(* Logix 5000 project; controller cal1632 1756-L62 rev 16.20; software revision 16.05; part 2 of 57 *)

ADD_ON_INSTRUCTION SYS_RPM_TO_SPEED   (* revision 1.0 *)
VAR_INPUT
   IN_gear_ratio : REAL; {required}
   IN_roll_diameter : REAL; {required}
   IN_vfd_fb_rpm : REAL; {required}
END_VAR
VAR_OUTPUT
   OUT_surface_speed_fb : REAL; {required}
END_VAR
VAR
   no_diameter : BOOL;
END_VAR

ROUTINE Logic   (* ladder *)
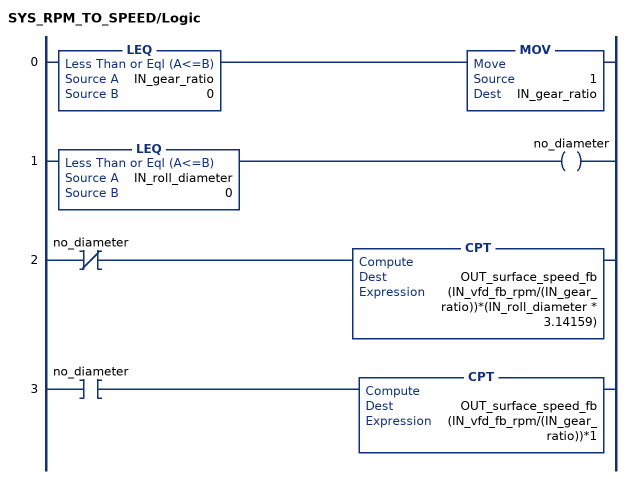
   0: LEQ(IN_gear_ratio,0)MOV(1,IN_gear_ratio);
   1: LEQ(IN_roll_diameter,0)OTE(no_diameter);
   2: XIO(no_diameter)CPT(OUT_surface_speed_fb,(IN_vfd_fb_rpm/(IN_gear_ratio))*(IN_roll_diameter * 3.14159));
   3: XIC(no_diameter)CPT(OUT_surface_speed_fb,(IN_vfd_fb_rpm/(IN_gear_ratio))*1);
END_ROUTINE
END_ADD_ON_INSTRUCTION

ADD_ON_INSTRUCTION SYS_SCP   (* revision 1.0 *)
VAR_INPUT
   Input : REAL; {required}
   Input_Min : REAL; {required}
   Input_Max : REAL; {required}
   Output_Min : REAL; {required}
   Output_Max : REAL; {required}
END_VAR
VAR_OUTPUT
   Output : REAL; {required}
   Fault : BOOL;
END_VAR
VAR
   m : REAL;
   b : REAL;
   X1 : REAL;
   X2 : REAL;
   Y1 : REAL;
   Y2 : REAL;
   X3 : REAL;
   Y3 : REAL;
END_VAR

ROUTINE Logic   (* ladder *)
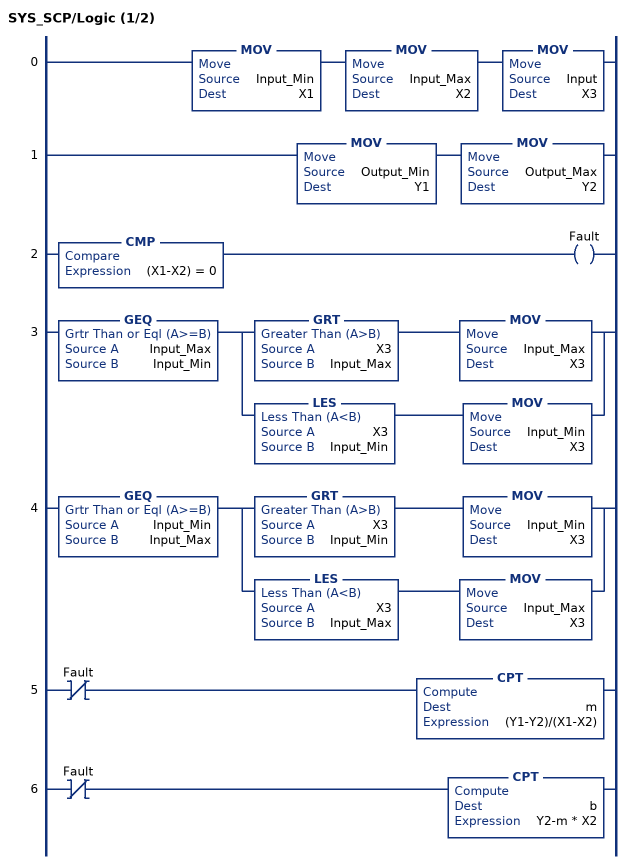
   0: MOV(Input_Min,X1)MOV(Input_Max,X2)MOV(Input,X3);
   1: MOV(Output_Min,Y1)MOV(Output_Max,Y2);
   2: CMP((X1-X2) = 0)OTE(Fault);
   3: GEQ(Input_Max,Input_Min)[GRT(X3,Input_Max) MOV(Input_Max,X3) ,LES(X3,Input_Min) MOV(Input_Min,X3) ];
   4: GEQ(Input_Min,Input_Max)[GRT(X3,Input_Min) MOV(Input_Min,X3) ,LES(X3,Input_Max) MOV(Input_Max,X3) ];
   5: XIO(Fault)CPT(m,(Y1-Y2)/(X1-X2));
   6: XIO(Fault)CPT(b,Y2-m * X2);
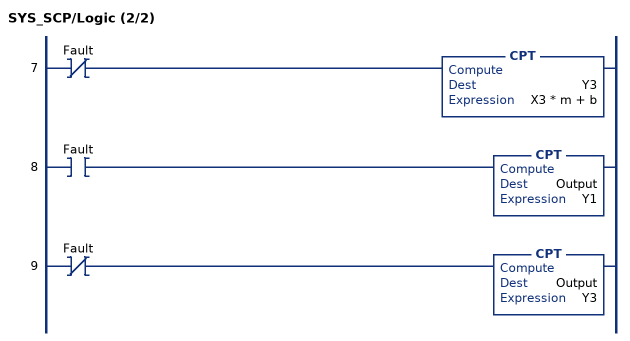
   7: XIO(Fault)CPT(Y3,X3 * m + b);
   8: XIC(Fault)CPT(Output,Y1);
   9: XIO(Fault)CPT(Output,Y3);
END_ROUTINE
END_ADD_ON_INSTRUCTION

ADD_ON_INSTRUCTION SYS_SPEED_TO_VFD   (* revision 1.0 *)
VAR_INPUT
   IN_gear_ratio : REAL; {required}
   IN_roll_diameter : REAL; {required}
   IN_selected_speed : REAL; {required}
END_VAR
VAR_OUTPUT
   OUT_surface_speed_rpm : REAL; {required}
END_VAR

ROUTINE Logic   (* ladder *)
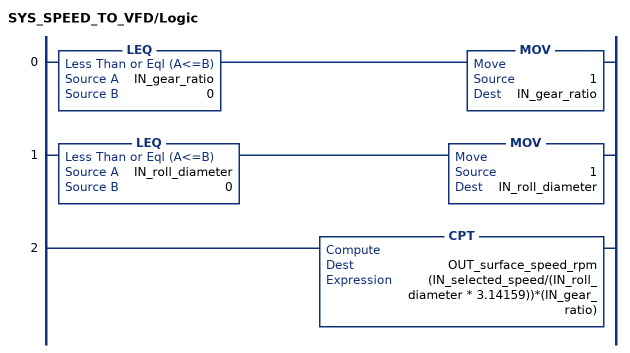
   0: LEQ(IN_gear_ratio,0)MOV(1,IN_gear_ratio);
   1: LEQ(IN_roll_diameter,0)MOV(1,IN_roll_diameter);
   2: CPT(OUT_surface_speed_rpm,(IN_selected_speed/(IN_roll_diameter * 3.14159))*(IN_gear_ratio));
END_ROUTINE
END_ADD_ON_INSTRUCTION

ADD_ON_INSTRUCTION SYS_Toggle   (* revision 1.0 *)
VAR_INPUT
   in_pb : BOOL; {required}
END_VAR
VAR_IN_OUT
   out_state : BOOL; {required}
END_VAR
VAR_INPUT
   toggle_state : BOOL; {visible}
END_VAR
VAR
   ons : DINT;
   toggle_select_deselct : BOOL;
END_VAR

ROUTINE Logic   (* ladder *)
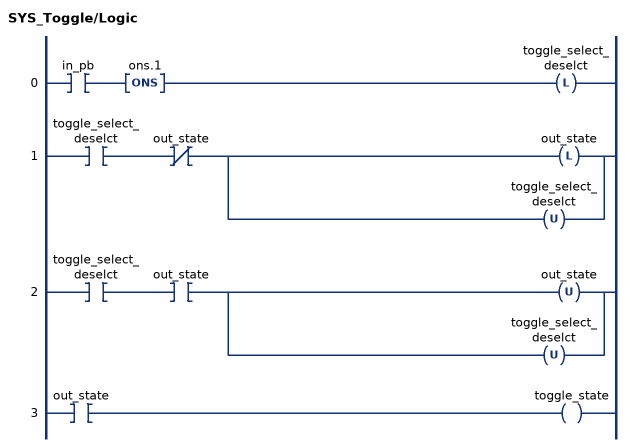
   0: XIC(in_pb)ONS(ons.1)OTL(toggle_select_deselct);
   1: XIC(toggle_select_deselct)XIO(out_state)[OTL(out_state) ,OTU(toggle_select_deselct) ];
   2: XIC(toggle_select_deselct)XIC(out_state)[OTU(out_state) ,OTU(toggle_select_deselct) ];
   3: XIC(out_state)OTE(toggle_state);
END_ROUTINE
END_ADD_ON_INSTRUCTION

VAR_GLOBAL   (* controller tags *)
   aaa_prs : REAL := 60.0;
   AFI : BOOL;
   FAULT : BOOL;
   HMI : BOOL;
   metering_roll : TIMER := (PRE := 4500);
   metering_roll_alarm : TIMER := (PRE := 4500);
   metering_roll_close : TIMER := (PRE := 5000);
   P00_VFD_Sprng_PID : PID := (SP := 25.0, OUT := 10.0);
   p01_ai_lc_4 : REAL := 0.95815146;
   p01_ai_prs : REAL := -2.5;
   p01_ai_tc : REAL := 132.4;
   p01_di_edge_ctrl_estop_active : BOOL;
   p01_di_estop_1_tripped : BOOL := 1;
   p01_di_estop_2_tripped : BOOL := 1;
   p01_di_estop_reset : BOOL;
   p01_di_impreg_estop_active : BOOL;
   p01_di_letoff_estop_active : BOOL;
   p01_di_lof_acc_estop_active : BOOL;
   p01_di_main_hmi_estop : BOOL;
   p01_di_rope_sw_1_active : BOOL;
   p01_di_rope_sw_2_active : BOOL;
   p01_di_rope_sw_3_active : BOOL;
   p01_di_rope_sw_4_active : BOOL;
   p01_di_rope_sw_5_active : BOOL;
   p01_di_rope_sw_6_active : BOOL;
   p01_di_rope_sw_7_active : BOOL;
   p01_di_rope_sw_8_active : BOOL;
   p01_di_splice_estop_active : BOOL;
   p01_di_ts2_estop_active : BOOL;
   p01_di_winder_estop_active : BOOL;
   p01_dint_to_hmi : DINT[16] := ([0] := 643, [1] := 2, [3] := 128, [4] := 2, [6] := 133, [7] := 2, [8] := 5, [9] := 9, [14] := 18806);
   p01_int_from_oxidizer : INT[10] := ([0] := 528, [1] := 2, [2] := 93, [3] := 121, [4] := 1688, [5] := 1689, [6] := 214, [7] := 88, [8] := 1385, [9] := 1608); {produced}
   p01_int_to_oxidizer : INT;
   p01_param_fan_zero_speed : REAL := 0.1;
   p01_param_heater_hl : REAL := 785.0;
   p01_param_master_accel : REAL := 0.5;
   p01_param_master_decel : REAL := 2.5;
   p01_param_master_jog_accel : REAL := 10.0;
   p01_param_master_jog_decel : REAL := 20.0;
   p01_param_master_jog_speed : REAL := 13.0;
   p01_param_min_start_tension : REAL := 10.0;
   p01_param_mtr_over_speed_pct : REAL := 0.4;
   p01_param_open_oven_exh_sp : REAL := 300.0;
   p01_param_open_oven_recirc_sp : REAL := 300.0;
   p01_param_open_oven_temp : REAL := 80.0;
   p01_param_oven_timer_presets : DINT[32] := ([1] := 500, [2] := 10000, [3] := 20000, [6] := 5000, [8] := 1000, [9] := 1000, [10] := 1000, [11] := 5000, [14] := 10000, [16] := 1000, [17] := 90000, [18] := 1500, [19] := 1000, [21] := 1000, [22] := 1000, [23] := 2000, [24] := 5000, [25] := 5000, [26] := 15000, [27] := 500, [28] := 30000, [31] := 500);
   p01_param_process_air_hl : REAL := 500.0;
   p01_param_process_air_max : REAL := 480.0;
   p01_param_slow_speed_sp : REAL := 2.0;
   p01_param_start_delay : REAL := 6.5;
   p01_param_temp_limit : REAL := 120.0;
   p01_param_tension_deviation : REAL := 5.0;
   p01_param_turret_dia_ft : REAL := 3.2;
   p01_r15_footage_ft : REAL;
   p01_real_to_hmi : REAL[112] := ([1] := 13.0, [11] := 92.0, [12] := 128.0, [13] := 1690.0, [14] := 1694.0, [15] := 220.0, [16] := 88.0, [17] := 1370.0, [18] := 1621.0, [19] := 8953.26);
   p01_recipe_active : recipe := (name := 'CP:F-555-S:1KPW:JOBY.csv', master_line_speed := 10.0, zone_1.recirc_sp := 1000.0, zone_1.exhaust_sp := 900.0, zone_1.temp_sp := 225.0, zone_2.recirc_sp := 1000.0, zone_2.exhaust_sp := 900.0, zone_2.temp_sp := 225.0, zone_3.recirc_sp := 1000.0, zone_3.exhaust_sp := 900.0, zone_3.temp_sp := 70.0, line_speed_sp := 13.0, letoff_tension_sp := 15.0, acc_tension_sp := 60.0, acc_fill_pressure_sp := 10.0, acc_counter_pressure_sp := 10.0, cure_time_sp := 55.0, platen_temp_sp := 450.0, impreg_gap_sp := 0.0175, impreg_supply_speed_sp := 1200.0, ts1_tension_sp := 60.0, adv_cooling_temp_sp := 65.0, ts2_tension_sp := 60.0, lower_poly_tension_sp := 3.0, lower_poly_b_tension_sp := 3.0, upper_poly_tension_sp := 3.0, upper_poly_b_tension_sp := 3.0, winder_tension_sp := 70.0, winder_torque_sp := 100.0, tension_deviation_sp := 15.0);
   p01_sys_enc : SYS_ENC := (IN_State := 3, OUT_Status := 1);
   p01_sys_lc : Limit_Clamp := (max := 100.0);
   p01_sys_scp : SYS_SCP := (Input := 12760.0, Input_Max := 30840.0, Output_Max := 50.0, Output := 20.68742);
   p01r01 : routine := (comment := 7);
   p01r02 : routine := (comment := -1073741569, fault := 32768, fault_ack := 32768);
   p01r02_all_fans_stopped : BOOL := 1;
   p01r02_batch_run_time : DINT := 24;
   p01r02_batch_run_time_hrs : DINT := 18806;
   p01r02_do_buzzer : BOOL;
   p01r02_do_buzzer_LINE : BOOL := 1;
   p01r02_do_green_stack_light_lel : BOOL := 1;
   p01r02_do_green_stack_light_LINE : BOOL;
   p01r02_do_horn : BOOL;
   p01r02_do_red_stack_light : BOOL;
   p01r02_do_red_stack_light_LINE : BOOL := 1;
   p01r02_do_yellow_stack_light : BOOL;
   p01r02_do_yellow_stack_light_LINE : BOOL := 1;
   p01r02_ethernet_comm : DINT := 491519;
   p01r02_fault_exists : BOOL;
   p01r02_flash_bit : BOOL;
   p01r02_flash_timer_off : TIMER := (PRE := 1000);
   p01r02_flash_timer_on : TIMER := (PRE := 1000, ACC := 979, EN := 1, TT := 1);
   p01r02_horn : BOOL := 1;
   p01r02_plc_faults : DINT := 16;
   p01r02_plc_scan_time : DINT := 30386;
   p01r02_plc_scan_time_in_sec : REAL := 0.030494;
   p01r02_timer_batch : TIMER := (PRE := 60000);
   p01r02_timer_fault : TIMER[25] := ([15].ACC := 31, [15].EN := 1, [15].DN := 1);
   p01r02_timer_half_second_off : TIMER := (PRE := 300);
   p01r02_timer_half_second_on : TIMER := (PRE := 300, ACC := 305, EN := 1, DN := 1);
   p01r02_timer_second : TIMER[2] := ([0].PRE := 1000, [0].ACC := 1009, [0].EN := 1, [0].DN := 1, [1].PRE := 1000, [1].ACC := 551, [1].EN := 1, [1].TT := 1);
   p01r02_timer_warning : TIMER[4];
   p01r02_unack_fault : BOOL;
   p01r02_unack_warning : BOOL := 1;
   p01r02_vfd_comm_2 : DINT[50] := ([0] := 16897, [1] := 16897, [2] := 16897, [3] := 16897, [4] := 16897, [5] := 16897, [6] := 16897, [7] := 16897, [8] := 16897, [9] := 16897, [10] := 16897, [11] := 16897, [12] := 16897, [13] := 16897, [14] := 16897, [15] := 4096, [16] := 16897, [17] := 16897, [18] := 16897);
   p01r02_warnings_exists : BOOL := 1;
   p01r03 : routine := (comment := -1073741793);
   p01r03_lc3_ave_ctrl : CONTROL := (LEN := 19);
   p01r03_oxidizer_prs : SYS_SCP := (Input_Max := 30840.0, Output_Min := -2.5, Output_Max := 2.5, Output := -2.5);
   p01r03_prs_input_max : REAL := 30840.0;
   p01r03_prs_input_min : REAL;
   p01r03_prs_output_max : REAL := 2.5;
   p01r03_prs_output_min : REAL := -2.5;
   p01r03_timer_fault : TIMER[4];
   p01r03_timer_warning : TIMER[4];
   p01r04 : routine := (comment := -1073741793);
   p01r04_LFL_warning : BOOL;
   p01r04_Temp_deviation_warning : BOOL := 1;
   p01r04_timer_fault : TIMER[4];
   p01r04_timer_warning : TIMER[4];
   p01r05 : routine := (comment := -1073741761);
   p01r05_enc : SYS_ENC;
   p01r05_timer_fault : TIMER[4];
   p01r05_timer_warning : TIMER[4];
   p01r06 : routine := (comment := -1073741572);
   p01r06_timer_fault : TIMER[4];
   p01r06_timer_warning : TIMER[4];
   p01r07 : routine := (comment := -1073741761);
   p01r07_timer_fault : TIMER[4];
   p01r07_timer_warning : TIMER[4];
   p01r08 : routine := (comment := -1073741761);
   p01r08_timer_fault : TIMER[4];
   p01r08_timer_warning : TIMER[4];
   p01r09 : routine := (comment := -1073741009, oneshot := 24, warning := 1, unack_warning := 1);
   p01r09_estop_ok : BOOL := 1;
   p01r09_mode_jog : BOOL;
   p01r09_mode_run : BOOL;
   p01r09_mode_thread : BOOL := 1;
   p01r09_open_oven : BOOL;
   p01r09_open_oven_toggle : SYS_Toggle;
   p01r09_pb_global_reset : BOOL;
   p01r09_pb_line_jog : BOOL;
   p01r09_permissive_change : BOOL;
   p01r09_request_line_jog : BOOL;
   p01r09_stretch_mode : BOOL;
   p01r09_timer_estop_reset : TIMER := (PRE := 1000, ACC := 1010, EN := 1, DN := 1);
   p01r09_timer_fault : TIMER[20];
   p01r09_timer_global_reset : TIMER := (PRE := 1000);
   p01r09_timer_warning : TIMER[4] := ([0].ACC := 31, [0].EN := 1, [0].DN := 1);
   p01r10 : routine := (comment := -1073741569);
   p01r10_fault_exists : BOOL := 1;
   p01r10_timer_fault : TIMER[4];
   p01r10_timer_warning : TIMER[4];
   p01r10_unack_fault : DINT := 12;
   p01r10_unack_fault_ex : BOOL := 1;
   p01r10_unack_warn_ex : BOOL := 1;
   p01r10_unack_warning : DINT := 15;
   p01r10_warning_exists : BOOL := 1;
   p01r11 : routine := (comment := -1073741761);
   p01r11_timer_fault : TIMER[4];
   p01r11_timer_warning : TIMER[4];
   p01r12 : routine := (comment := -1073741761);
   p01r12_accel_rate : REAL := 0.5;
   p01r12_decel_rate : REAL := 2.5;
   p01r12_line_at_speed : BOOL;
   p01r12_master_acel_decel_ramp : SYS_ACC_DEC_RAMP := (IN_param_master_accel_rate := 0.5, IN_param_master_decel_rate := 2.5, IN_last_scan_s := 0.03063);
   p01r12_master_ramped_speed : REAL;
   p01r12_ramped_setpoint : REAL;
   p01r12_request_any_jog_thread : BOOL;
   p01r12_selected_line_speed : REAL;
   p01r12_timer_fault : TIMER[8];
   p01r12_timer_warning : TIMER[8];
   p01r12_zero_line_speed : BOOL := 1;
   p01r13 : routine := (comment := -1073708945);
   p01r13_check_status : BOOL;
   p01r13_check_status_time : REAL := 6250.0;
   p01r13_check_status_timer : TIMER := (PRE := 15000);
   p01r13_check_tension : TIMER;
   p01r13_letoff_tension_ok : BOOL;
   p01r13_LFL_stop : BOOL;
   p01r13_line_running : BOOL;
   p01r13_line_slow_ramp : BOOL;
   p01r13_line_start : SYS_ENC := (IN_State := 513, OUT_Status := 9);
   p01r13_oven_temp_ok : BOOL;
   p01r13_pb_start : BOOL;
   p01r13_pb_stop : BOOL;
   p01r13_permissive_drives : BOOL;
   p01r13_permissive_line_run : BOOL;
   p01r13_permissive_oven : BOOL := 1;
   p01r13_permissive_oxidizer : BOOL;
   p01r13_request_run : BOOL;
   p01r13_request_stop : BOOL := 1;
   p01r13_state : DINT := 513;
   p01r13_status : DINT := 9;
   p01r13_system_mode_run : BOOL;
   p01r13_temperature_status_check : TIMER := (PRE := 10000);
   p01r13_tension_ok : BOOL;
   p01r13_timer_fault : TIMER[8];
   p01r13_timer_line_start_warning_dwell : TIMER := (PRE := 6500);
   p01r13_timer_line_stop_dwell : TIMER := (PRE := 60000);
   p01r13_timer_switch_to_stretch_dwell : TIMER;
   p01r13_timer_warning : TIMER[8];
   p01r13_ts1_tension_ok : BOOL;
   p01r13_ts2_tension_ok : BOOL;
   p01r13_winder_tension_ok : BOOL;
   p01r14 : routine := (comment := -1073741697);
   p01r14_msg_read : MESSAGE;
        MessageParameters(ServiceCode := 16#0fa2, LocalElement := p01_int_from_oxidizer[0], ...)
   p01r14_msg_read_retry_timer : TIMER := (PRE := 1000);
   p01r14_msg_read_timer : TIMER := (PRE := 200, ACC := 61, EN := 1, TT := 1);
   p01r14_msg_write : MESSAGE;
        MessageParameters(ServiceCode := 16#0faa, LocalElement := p01_int_to_oxidizer, ...)
   p01r14_msg_write_retry_timer : TIMER := (PRE := 1000);
   p01r14_msg_write_timer : TIMER := (PRE := 100, EN := 1, TT := 1);
   p01r14_oxidizer_heart_beat_off : TIMER := (PRE := 4000);
   p01r14_oxidizer_heart_beat_ok : BOOL := 1;
   p01r14_oxidizer_heart_beat_on : TIMER := (PRE := 4000);
   p01r14_oxidizer_mass_flow : REAL := 8947.989;
   p01r14_timer_fault : TIMER[10] := ([1].PRE := 2000, [2].PRE := 1000);
   p01r14_timer_warning : TIMER[5];
   p02_dint_from_hmi : hmi_dint := (zone_3[6] := 256);
   p02_dint_to_hmi : hmi_dint := (global[0] := 643, global[1] := 2, global[3] := 128, global[4] := 2, global[6] := 133, global[7] := 2, global[8] := 5, global[9] := 9, global[14] := 18806, zone_1[2] := 1114304, zone_1[4] := 656995, zone_1[5] := 5793, zone_1[6] := 28784, zone_1[8] := 2, zone_1[9] := 4, zone_1[10] := 3, zone_1[11] := 3, zone_2[2] := 1114240, zone_2[4] := 656995, zone_2[5] := 9889, zone_2[6] := 28784, zone_2[8] := 2, zone_2[9] := 4, zone_2[10] := 3, zone_2[11] := 3, zone_3[4] := 655971, zone_3[5] := 1060, zone_3[6] := 28784, zone_3[8] := 1, zone_3[9] := 1, zone_3[10] := 3, zone_3[11] := 3, letoff[0] := 38, letoff[1] := 7368816, letoff[2] := 320, letoff[4] := 48, letoff[6] := 131072, letoff[7] := 1, ts1[0] := 4, ts1[1] := 4920, ts1[2] := 5, ts1[7] := 2, ts2[0] := 983808, ts2[1] := 4920, ts2[2] := 5, ts2[6] := 131072, ts2[7] := 2, upl[0] := 5, lpl[0] := 4, wdr[0] := 4, wdr[1] := 4920, wdr[2] := 1285, wdr[3] := 4920, wdr[4] := 512, wdr[5] := 112, splice[10] := 2, edg[0] := 1, slt[0] := 4, slt[1] := 1024, impreg[1] := 33845488,
        impreg[3] := 207668736, impreg[4] := 4352, impreg[5] := 2, impreg[6] := 2, impreg[7] := 3, impreg[10] := -1, impreg[11] := -1, impreg[12] := -1, impreg[13] := -1, adv_cooling[0] := 655360, adv_cooling[1] := 32768, adv_cooling[5] := 16382, retraction[0] := 255);
   p02_real_from_hmi : hmi_real := (global[1] := 13.0, zone_1[39] := 5.0, zone_1[44] := 50.0, zone_1[47] := 15.0, zone_1[48] := 20.0, zone_1[49] := 2.0, zone_1[51] := 15.0, zone_1[52] := 440.0, zone_1[54] := 20.0, zone_1[55] := 25.0, zone_1[56] := 40.0, zone_1[57] := 110.0, zone_1[58] := -0.25, zone_1[59] := 20.0, zone_1[60] := 20.0, zone_1[68] := 50.0, zone_2[39] := 5.0, zone_2[44] := 50.0, zone_2[47] := 15.0, zone_2[48] := 25.0, zone_2[49] := 2.0, zone_2[51] := 15.0, zone_2[52] := 440.0, zone_2[54] := 20.0, zone_2[55] := 25.0, zone_2[56] := 40.0, zone_2[57] := 110.0, zone_2[58] := -0.25, zone_2[59] := 15.0, zone_2[60] := 20.0, zone_2[68] := 15.0, zone_3[39] := 5.0, zone_3[44] := 10.0, zone_3[45] := 0.1, zone_3[48] := 75.0, zone_3[49] := 0.22, zone_3[52] := 400.0, zone_3[54] := 25.0, zone_3[55] := 25.0, zone_3[56] := 40.0, zone_3[57] := 125.0, zone_3[59] := 5.0, zone_3[60] := 15.0, zone_3[68] := 100.0, letoff[40] := 1.8, letoff[41] := 2.0, letoff[43] := 0.01, ts1[40] := 5.0, ts1[41] := 2.0, ts2[40] := 3.2, ts2[41] := 0.5, wdr[40] := 0.75, wdr[41] := 0.8, wdr[60] := 100.0, wdr[61] := 100.0, splice[44] := 30.0, splice[47] := 30.0, impreg[0] := 0.014, impreg[1] := 0.014, impreg[2] := 0.003,
        impreg[3] := 0.0145, impreg[55] := 10.0, impreg[56] := 30.0, impreg[58] := -0.25, adv_cooling[48] := 50.0, adv_cooling[49] := 1.0, adv_cooling[54] := 20.0, adv_cooling[58] := 10.0, adv_cooling[66] := 15.0, adv_cooling[68] := 100.0);
   p02_real_to_hmi : hmi_real := (global[1] := 13.0, global[11] := 92.0, global[12] := 105.0, global[13] := 1664.0, global[14] := 1675.0, global[15] := 197.0, global[16] := 88.0, global[17] := 1369.0, global[18] := 1614.0, global[19] := 8963.069, zone_1[0] := 181.90001, zone_1[1] := 181.7, zone_1[2] := 181.90001, zone_1[6] := -0.08177692, zone_1[8] := 3.8146973e-06, zone_1[12] := 3.8146973e-06, zone_1[44] := 50.0, zone_1[47] := 15.0, zone_1[48] := 20.0, zone_1[49] := 2.0, zone_1[51] := 15.0, zone_1[52] := 440.0, zone_1[54] := 20.0, zone_1[55] := 25.0, zone_1[56] := 40.0, zone_1[57] := 110.0, zone_1[58] := -0.25, zone_1[59] := 20.0, zone_1[60] := 20.0, zone_1[67] := 225.0, zone_1[68] := 50.0, zone_1[72] := 181.90001, zone_2[0] := 196.3, zone_2[1] := 197.40001, zone_2[2] := 196.3, zone_2[6] := 0.0044070184, zone_2[8] := 3.8146973e-06, zone_2[12] := 3.8146973e-06, zone_2[44] := 50.0, zone_2[47] := 15.0, zone_2[48] := 25.0, zone_2[49] := 2.0, zone_2[51] := 15.0, zone_2[52] := 440.0, zone_2[54] := 20.0, zone_2[55] := 25.0, zone_2[56] := 40.0, zone_2[57] := 110.0, zone_2[58] := -0.25, zone_2[59] := 15.0, zone_2[60] := 20.0, zone_2[67] := 225.0, zone_2[68] := 15.0, zone_2[72] := 196.3, zone_3[0] := 67.200005, zone_3[1] := 65.6, zone_3[2] := 67.200005, zone_3[8] := 3.8146973e-06, zone_3[12] := 3.8146973e-06, zone_3[44] := 10.0,
        zone_3[45] := 0.1, zone_3[48] := 75.0, zone_3[49] := 0.22, zone_3[52] := 400.0, zone_3[54] := 25.0, zone_3[55] := 25.0, zone_3[56] := 40.0, zone_3[57] := 125.0, zone_3[59] := 5.0, zone_3[60] := 15.0, zone_3[67] := 70.0, zone_3[68] := 100.0, zone_3[72] := 67.200005, letoff[0] := 0.9617673, letoff[1] := 23.62944, letoff[2] := 0.18760681, letoff[8] := 3.8146973e-06, letoff[14] := -3.8146973e-06, letoff[15] := 65.0, letoff[20] := -3.8146973e-06, letoff[22] := 17.604113, letoff[25] := 10.0, letoff[26] := 32.0, letoff[27] := 32.0, letoff[40] := 1.8, letoff[41] := 2.0, ts1[0] := 13.29894, ts1[40] := 5.0, ts1[41] := 2.0, ts2[40] := 3.2, ts2[41] := 0.5, upl[0] := -75.37109, upl[1] := -85.5, lpl[0] := -38.8816, lpl[1] := 8.07605, wdr[0] := 72.75, wdr[1] := 21.514273, wdr[3] := 8.401376, wdr[4] := 7.487962, wdr[21] := 9.277759, wdr[40] := 0.75, wdr[41] := 0.8, splice[0] := 365.9, splice[1] := 55.0, impreg[0] := 0.014, impreg[1] := 0.014, impreg[2] := 0.003, impreg[3] := 0.0145, impreg[8] := 3.8146973e-06, impreg[11] := 60.0, impreg[17] := 6553.3003, impreg[22] := 0.008, impreg[23] := 65532.0, impreg[28] := -0.0032749623, impreg[55] := 10.0, impreg[56] := 30.0, impreg[58] := -0.25, impreg[60] := 0.008, impreg[61] := 0.008, slt[7] := -3.8146973e-06,
        adv_cooling[0] := 65.6, adv_cooling[1] := 2192.0, adv_cooling[2] := 65.6, adv_cooling[6] := 14.68742, adv_cooling[48] := 50.0, adv_cooling[49] := 1.0, adv_cooling[54] := 20.0, adv_cooling[58] := 10.0, adv_cooling[68] := 100.0, adv_cooling[72] := 65.6, adv_cooling[80] := -1.22e-43, adv_cooling[81] := -1.e-44, adv_cooling[82] := 2.120817e-38, adv_cooling[83] := 5.91931e-40, adv_cooling[84] := -1.471751e-20, adv_cooling[85] := 1.e-45, adv_cooling[87] := -1.e-44, adv_cooling[88] := -1.e-44, adv_cooling[89] := 2.120817e-38, adv_cooling[90] := 4.14325e-40, adv_cooling[91] := 1.4850275e+36, adv_cooling[92] := 1.e-45, adv_cooling[94] := -1.e-44, adv_cooling[95] := -2.2e-44, adv_cooling[96] := 2.120817e-38, adv_cooling[97] := 5.70777e-40, adv_cooling[98] := -2.1817042e+21, adv_cooling[99] := 5.6e-44, adv_cooling[100] := -2.00006, adv_cooling[110] := -2.2e-44, adv_cooling[111] := -1.e-44);
   p02_recipe_from_hmi : recipe := (name := 'CP:F-555-S:1KPW:JOBY.csv', master_line_speed := 10.0, zone_1.recirc_sp := 1000.0, zone_1.exhaust_sp := 900.0, zone_1.temp_sp := 225.0, zone_2.recirc_sp := 1000.0, zone_2.exhaust_sp := 900.0, zone_2.temp_sp := 225.0, zone_3.recirc_sp := 1000.0, zone_3.exhaust_sp := 900.0, zone_3.temp_sp := 70.0, line_speed_sp := 13.0, letoff_tension_sp := 15.0, acc_tension_sp := 60.0, acc_fill_pressure_sp := 10.0, acc_counter_pressure_sp := 10.0, cure_time_sp := 55.0, platen_temp_sp := 450.0, impreg_gap_sp := 0.0175, impreg_supply_speed_sp := 1200.0, ts1_tension_sp := 60.0, adv_cooling_temp_sp := 65.0, ts2_tension_sp := 60.0, lower_poly_tension_sp := 3.0, lower_poly_b_tension_sp := 3.0, upper_poly_tension_sp := 3.0, upper_poly_b_tension_sp := 3.0, winder_tension_sp := 70.0, winder_torque_sp := 100.0, tension_deviation_sp := 15.0);
   p02_recipe_to_hmi : recipe := (name := 'CP:F-555-S:1KPW:JOBY.csv', master_line_speed := 10.0, zone_1.recirc_sp := 1000.0, zone_1.exhaust_sp := 900.0, zone_1.temp_sp := 225.0, zone_2.recirc_sp := 1000.0, zone_2.exhaust_sp := 900.0, zone_2.temp_sp := 225.0, zone_3.recirc_sp := 1000.0, zone_3.exhaust_sp := 900.0, zone_3.temp_sp := 70.0, line_speed_sp := 13.0, letoff_tension_sp := 15.0, acc_tension_sp := 60.0, acc_fill_pressure_sp := 10.0, acc_counter_pressure_sp := 10.0, cure_time_sp := 55.0, platen_temp_sp := 450.0, impreg_gap_sp := 0.0175, impreg_supply_speed_sp := 1200.0, ts1_tension_sp := 60.0, adv_cooling_temp_sp := 65.0, ts2_tension_sp := 60.0, lower_poly_tension_sp := 3.0, lower_poly_b_tension_sp := 3.0, upper_poly_tension_sp := 3.0, upper_poly_b_tension_sp := 3.0, winder_tension_sp := 70.0, winder_torque_sp := 100.0, tension_deviation_sp := 15.0);
   p02r01 : routine := (comment := 7);
   p02r02 : routine := (comment := -1073741761, oneshot := 1);
   p02r02_timer_fault : TIMER[4];
   p02r02_timer_logout : TIMER := (PRE := 900000, ACC := 900000);
   p02r02_timer_warning : TIMER[4];
   p02r03 : routine := (comment := -1073741793);
   p02r03_timer_fault : TIMER[4];
   p02r03_timer_warning : TIMER[4];
   p02r04 : routine := (comment := -536870835);
   p02r04_timer_fault : TIMER[4];
   p02r04_timer_warning : TIMER[4];
   p02r05 : routine := (comment := -1073741729);
   p02r05_timer_fault : TIMER[4];
   p02r05_timer_warning : TIMER[4];
   p02r06 : routine := (comment := -1073737569);
   p02r06_timer_fault : TIMER[4];
   p02r06_timer_warning : TIMER[4];
   p02r07 : routine := (comment := -1073737721);
   p02r07_timer_fault : TIMER[4];
   p02r07_timer_warning : TIMER[4];
   p02r08 : routine := (comment := -1073741817);
   p02r08_timer_fault : TIMER[4];
   p02r08_timer_warning : TIMER[4];
   p02r09 : routine := (comment := -1073741761);
   p02r09_timer_fault : TIMER[4];
   p02r09_timer_warning : TIMER[4];
   p02r10 : routine := (comment := -1073741761);
   p02r10_timer_fault : TIMER[4];
   p02r10_timer_warning : TIMER[4];
   p02r11 : routine := (comment := -1073741761);
   p02r11_timer_fault : TIMER[4];
   p02r11_timer_warning : TIMER[4];
   p02r12 : routine := (comment := -1073741761);
   p02r12_timer_fault : TIMER[4];
   p02r12_timer_warning : TIMER[4];
   p02r13 : routine := (comment := -1073741761);
   p02r13_timer_fault : TIMER[4];
   p02r13_timer_warning : TIMER[4];
   p02r14 : routine := (comment := -1073741761);
   p02r14_timer_fault : TIMER[4];
   p02r14_timer_warning : TIMER[4];
   p02r15 : routine := (comment := -1073741761);
   p02r15_timer_fault : TIMER[4];
   p02r15_timer_warning : TIMER[4];
   p11_ai_exh_amps : REAL;
   p11_ai_exh_hz : REAL := 3.8146973e-06;
   p11_ai_exh_hz_max : REAL := 60.0;
   p11_ai_exh_pct : REAL;
   p11_ai_exh_rpm : REAL;
   p11_ai_lfl : REAL;
   p11_ai_prs : REAL := -0.080804154;
   p11_ai_recirc_amps : REAL;
   p11_ai_recirc_hz : REAL := 3.8146973e-06;
   p11_ai_recirc_hz_max : REAL := 60.0;
   p11_ai_recirc_pct : REAL;
   p11_ai_recirc_rpm : REAL;
   p11_ai_tc01 : REAL := 183.5;
   p11_ai_tc02 : REAL := 183.5;
   p11_ao_cv : REAL;
   p11_ao_exhaust_selected_speed : REAL;
   p11_ao_recirc_selected_speed : REAL;
   p11_di_burner_auto : BOOL := 1;
   p11_di_burner_safeties_ok : BOOL;
   p11_di_door_open : BOOL;
   p11_di_exh : acs800_di_normal := (ready := 1, ctrl_from_net := 1, ref_from_net := 1);
   p11_di_exh_fan_mtr_ts : BOOL := 1;
   p11_di_exh_flow_ok : BOOL;
   p11_di_flame_failure : BOOL;
   p11_di_flame_on : BOOL;
   p11_di_fresh_air_clean : BOOL;
   p11_di_high_limit_temp_ok : BOOL := 1;
   p11_di_recirc : acs800_di_normal := (ready := 1, ctrl_from_net := 1, ref_from_net := 1);
   p11_di_recirc_fan_mtr_ts : BOOL := 1;
   p11_di_recirc_flow_ok : BOOL;
   p11_di_sp0 : BOOL;
   p11_di_sp00 : BOOL;
   p11_di_sp1 : BOOL;
   p11_di_sp2 : BOOL;
   p11_di_sp3 : BOOL;
   p11_di_tc01_bo : BOOL;
   p11_di_tc02_bo : BOOL;
   p11_di_zone_air_clean : BOOL;
   p11_dint_to_hmi : DINT[16] := ([2] := 1114304, [4] := 656995, [5] := 5793, [6] := 28784, [8] := 2, [9] := 4, [10] := 3, [11] := 3);
   p11_do_enable_burner : BOOL;
   p11_do_exh : acs800_do_normal;
   p11_do_recirc : acs800_do_normal;
   p11_do_rst_flame : BOOL;
   p11_exhaust_input_max : REAL := 2000.0;
   p11_exhaust_input_min : REAL;
   p11_exhaust_output_max : REAL := 2000.0;
   p11_exhaust_output_min : REAL;
   p11_hc_input_max : REAL := 100.0;
   p11_hc_input_min : REAL;
   p11_hc_output_max : REAL := 30840.0;
   p11_hc_output_min : REAL;
   p11_lfl_input_max : REAL := 30840.0;
   p11_lfl_input_min : REAL;
   p11_lfl_output_max : REAL := 100.0;
   p11_lfl_output_min : REAL;
   p11_param_fast_to_soak : REAL := 20.0;
   p11_param_lfl_hhl : REAL := 40.0;
   p11_param_lfl_hl : REAL := 25.0;
   p11_param_pid1_ff : REAL := 15.0;
   p11_param_pid1_kd : REAL;
   p11_param_pid1_ki : REAL;
   p11_param_pid1_kp : REAL := 50.0;
   p11_param_pid2_ff : REAL := 15.0;
   p11_param_pid2_kd : REAL;
   p11_param_pid2_ki : REAL := 2.0;
   p11_param_pid2_kp : REAL := 20.0;
   p11_param_shutdown_temp : REAL := 110.0;
   p11_param_soak_to_fast : REAL := 20.0;
   p11_param_tc01_dev : REAL := 20.0;
   p11_param_tc01_hl : REAL := 440.0;
   p11_param_tc01z : REAL;
   p11_param_tc02z : REAL;
   p11_param_zone_pressure : REAL := -0.25;
   p11_prs_input_max : REAL := 30840.0;
   p11_prs_input_min : REAL;
   p11_prs_output_max : REAL := 0.25;
   p11_prs_output_min : REAL := -0.25;
   p11_real_to_hmi : REAL[112] := ([0] := 182.3, [1] := 182.1, [2] := 182.3, [6] := -0.08305772, [8] := 3.8146973e-06, [12] := 3.8146973e-06, [44] := 50.0, [47] := 15.0, [48] := 20.0, [49] := 2.0, [51] := 15.0, [52] := 440.0, [54] := 20.0, [55] := 25.0, [56] := 40.0, [57] := 110.0, [58] := -0.25, [59] := 20.0, [60] := 20.0, [67] := 225.0, [68] := 50.0, [72] := 182.3);
   p11_recirc_input_max : REAL := 2000.0;
   p11_recirc_input_min : REAL;
   p11_recirc_output_max : REAL := 2000.0;
   p11_recirc_output_min : REAL;
   p11r01 : routine := (comment := 7);
   p11r02 : routine := (comment := -1073741761);
   p11r02_fault_exists : BOOL;
   p11r02_not_safe_temp : BOOL := 1;
   p11r02_safe_temp : BOOL;
   p11r02_shutdown_temp : BOOL;
   p11r02_timer_fault : TIMER[4];
   p11r02_timer_safe_temp : TIMER[2] := ([0].PRE := 30000, [1].PRE := 30000, [1].ACC := 30014, [1].EN := 1, [1].DN := 1);
   p11r02_timer_warning : TIMER[4] := ([0].PRE := 1500);
   p11r02_unack_fault : BOOL;
   p11r02_unack_warning : BOOL := 1;
   p11r02_warning_exists : BOOL := 1;
   p11r03 : routine := (comment := -1073741761);
   p11r03_hz : SYS_SCP := (Input_Max := 1750.0, Output_Max := 60.0, Output := 3.8146973e-06);
   p11r03_timer_fault : TIMER[4];
   p11r03_timer_warning : TIMER[4];
   p11r04 : routine := (comment := -1073741761);
   p11r04_timer_fault : TIMER[4];
   p11r04_timer_warning : TIMER[4];
   p11r05 : routine := (comment := -1073741761, state := 7);
   p11r05_exh_status : DINT := 3;
   p11r05_recirc_status : DINT := 3;
   p11r05_temp_ctrl_status : DINT := 4;
   p11r05_timer_fault : TIMER[4];
   p11r05_timer_warning : TIMER[4];
   p11r06 : routine := (comment := -1073741572);
   p11r06_timer_fault : TIMER[4];
   p11r06_timer_warning : TIMER[4];
   p11r07 : routine := (comment := -1073741761);
   p11r07_timer_fault : TIMER[4];
   p11r07_timer_warning : TIMER[4];
   p11r08 : routine := (comment := -1073741761);
   p11r08_timer_fault : TIMER[4];
   p11r08_timer_warning : TIMER[4];
   p11r09 : routine := (comment := -1073741761);
   p11r09_timer_fault : TIMER[4];
   p11r09_timer_warning : TIMER[8];
   p11r10 : routine := (comment := -1073741761);
   p11r10_timer_fault : TIMER[4];
   p11r10_timer_warning : TIMER[4];
   p11r12_Oven_auto_run_on : BOOL;
   p11r16_pid_temp_cv : DINT;
   p11r16_temp_ok : BOOL := 1;
   p11r20 : routine := (comment := -1073741761);
   p11r20_safeties_ok : BOOL;
   p11r20_state : DINT := 5;
   p11r20_status : DINT := 2;
   p11r20_timer_fault : TIMER[4];
   p11r20_timer_state_11 : TIMER := (PRE := 5000, ACC := 5019, EN := 1, DN := 1);
   p11r20_timer_state_3 : TIMER := (PRE := 1000);
   p11r20_timer_state_4 : TIMER := (PRE := 1000);
   p11r20_timer_state_7 : TIMER := (PRE := 2000);
   p11r20_timer_warning : TIMER[4];
   p11r30 : routine := (comment := -1073741697, warning := 192, warning_ack := 192);
   p11r30_cv_man_sp : REAL := 50.0;
   p11r30_pb_auto : BOOL;
   p11r30_pb_manual : BOOL;
   p11r30_pb_zone_off : BOOL;
   p11r30_pb_zone_on : BOOL;
   p11r30_permissive_run : BOOL;
   p11r30_pid_temp : PID := (CTL := -2077195136, EN := 1, SWM := 1, NOBC := 1, NOZC := 1, INI := 1, DVNA := 1, PVHA := 1, KP := 20.0, KI := 2.0, BIAS := 15.0, MAXS := 1000.0, MAXO := 100.0, UPD := 0.01, PV := 182.8, ERR := -182.8, MAXI := 10000.0, MAXCV := 100.0, MAXTIE := 100.0, DATA[0] := 350.6, DATA[1] := -292.48, DATA[2] := 182.8, DATA[3] := -182.8, DATA[5] := 0.1, DATA[6] := 0.1, DATA[7] := 0.16, DATA[8] := 20.0, DATA[9] := 2.0, DATA[11] := 20.0, DATA[12] := 2.0, DATA[15] := 1.0, DATA[16] := 1.0);
   p11r30_pid_temp_pv : REAL := 1823.0;
   p11r30_pid_temp_sp : REAL := 225.0;
   p11r30_pid_temp_sp_error : REAL := 183.2;
   p11r30_pid_temp_sp_last : REAL := 225.0;
   p11r30_request_deviation_warning : BOOL;
   p11r30_request_heat : BOOL;
   p11r30_request_heat_last : BOOL;
   p11r30_request_manual : BOOL;
   p11r30_request_PID_shot : BOOL;
   p11r30_request_soak_control : BOOL := 1;
   p11r30_temp_deviation_setpoint : DINT := 5;
   p11r30_timer_fault : TIMER[16] := ([0].PRE := 5000, [2].PRE := 1000, [4].PRE := 1000, [10].PRE := 5000, [11].PRE := 5000, [12].PRE := 5000);
   p11r30_timer_warning : TIMER[12] := ([0].PRE := 10000, [1].PRE := 1000, [2].PRE := 1000, [3].PRE := 90000, [4].PRE := 1000, [6].PRE := 1000, [6].ACC := 1010, [6].EN := 1, [6].DN := 1, [7].PRE := 1000, [7].ACC := 1010, [7].EN := 1, [7].DN := 1, [8].PRE := 1000);
   p11r30_vfds_ok : BOOL;
   p11r30_vfds_ready : BOOL := 1;
   p11r31 : routine := (comment := -1073741697, warning := 1, unack_warning := 1);
   p11r31_pb_start : BOOL;
   p11r31_pb_stop : BOOL;
   p11r31_request_auto_run : BOOL;
   p11r31_request_auto_stop : BOOL := 1;
   p11r31_run_permissive : BOOL := 1;
   p11r31_timer_fault : TIMER[5] := ([1].PRE := 500);
   p11r31_timer_prs : TIMER := (PRE := 2500);
   p11r31_timer_warning : TIMER[5] := ([0].PRE := 10000, [0].ACC := 10014, [0].EN := 1, [0].DN := 1, [1].PRE := 20000, [2].PRE := 500);
   p11r31_vfd_stopped : BOOL := 1;
   p11r32 : routine := (comment := -536870849, warning := 1, unack_warning := 1);
   p11r32_pb_start : BOOL;
   p11r32_pb_stop : BOOL;
   p11r32_request_auto_run : BOOL;
   p11r32_request_auto_stop : BOOL := 1;
   p11r32_run_permissive : BOOL := 1;
   p11r32_timer_fault : TIMER[5] := ([1].PRE := 500);
   p11r32_timer_warning : TIMER[5] := ([0].PRE := 10000, [0].ACC := 10014, [0].EN := 1, [0].DN := 1, [1].PRE := 20000, [2].PRE := 20000);
   p11r32_vfd_stopped : BOOL := 1;
   p12_ai_exhaust_amps : REAL;
   p12_ai_exhaust_hz : REAL := 3.8146973e-06;
   p12_ai_exhaust_hz_max : REAL := 60.0;
   p12_ai_exhaust_pct : REAL;
   p12_ai_exhaust_rpm : REAL;
   p12_ai_lfl : REAL;
   p12_ai_prs : REAL := 0.0023331344;
   p12_ai_recirc_amps : REAL;
   p12_ai_recirc_hz : REAL := 3.8146973e-06;
   p12_ai_recirc_hz_max : REAL := 60.0;
   p12_ai_recirc_pct : REAL;
   p12_ai_recirc_rpm : REAL;
   p12_ai_tc01 : REAL := 197.6;
   p12_ai_tc02 : REAL := 197.2;
   p12_ao_cv : REAL;
   p12_ao_exhaust_selected_speed : REAL;
   p12_ao_recirc_selected_speed : REAL;
   p12_di_burner_auto : BOOL := 1;
   p12_di_burner_safeties_ok : BOOL;
   p12_di_door_open : BOOL;
   p12_di_exh : acs800_di_normal := (ready := 1, ctrl_from_net := 1, ref_from_net := 1);
   p12_di_exh_fan_mtr_ts : BOOL := 1;
   p12_di_exh_flow_ok : BOOL;
   p12_di_flame_failure : BOOL;
   p12_di_flame_on : BOOL;
   p12_di_fresh_air_clean : BOOL := 1;
   p12_di_high_limit_temp_ok : BOOL := 1;
   p12_di_recirc : acs800_di_normal := (ready := 1, ctrl_from_net := 1, ref_from_net := 1);
   p12_di_recirc_fan_mtr_ts : BOOL := 1;
   p12_di_recirc_flow_ok : BOOL;
   p12_di_sp0 : BOOL;
   p12_di_sp00 : BOOL;
   p12_di_sp1 : BOOL;
   p12_di_sp2 : BOOL;
   p12_di_sp3 : BOOL;
   p12_di_tc01_bo : BOOL;
   p12_di_tc02_bo : BOOL;
   p12_di_zone_air_clean : BOOL;
   p12_dint_to_hmi : DINT[16] := ([2] := 1114240, [4] := 656995, [5] := 9889, [6] := 28784, [8] := 2, [9] := 4, [10] := 3, [11] := 3);
   p12_do_enable_burner : BOOL;
   p12_do_exh : acs800_do_normal;
   p12_do_recirc : acs800_do_normal;
   p12_do_rst_flame : BOOL;
   p12_exhaust_input_max : REAL := 2000.0;
   p12_exhaust_input_min : REAL;
   p12_exhaust_output_max : REAL := 2000.0;
   p12_exhaust_output_min : REAL;
   p12_hc_input_max : REAL := 100.0;
   p12_hc_input_min : REAL;
   p12_hc_output_max : REAL := 30840.0;
   p12_hc_output_min : REAL;
   p12_lfl_input_max : REAL := 30840.0;
   p12_lfl_input_min : REAL;
   p12_lfl_output_max : REAL := 100.0;
   p12_lfl_output_min : REAL;
   p12_param_fast_to_soak : REAL := 15.0;
   p12_param_lfl_hhl : REAL := 40.0;
   p12_param_lfl_hl : REAL := 25.0;
   p12_param_pid1_ff : REAL := 15.0;
   p12_param_pid1_kd : REAL;
   p12_param_pid1_ki : REAL;
   p12_param_pid1_kp : REAL := 50.0;
   p12_param_pid2_ff : REAL := 15.0;
   p12_param_pid2_kd : REAL;
   p12_param_pid2_ki : REAL := 2.0;
   p12_param_pid2_kp : REAL := 25.0;
   p12_param_shutdown_temp : REAL := 110.0;
   p12_param_soak_to_fast : REAL := 20.0;
   p12_param_tc01_dev : REAL := 20.0;
   p12_param_tc01_hl : REAL := 440.0;
   p12_param_tc01z : REAL;
   p12_param_tc02z : REAL;
   p12_param_zone_pressure : REAL := -0.25;
   p12_prs_input_max : REAL := 30860.0;
   p12_prs_input_min : REAL;
   p12_prs_output_max : REAL := 0.25;
   p12_prs_output_min : REAL := -0.25;
   p12_real_to_hmi : REAL[112] := ([0] := 197.40001, [1] := 197.90001, [2] := 197.40001, [6] := 0.0036131144, [8] := 3.8146973e-06, [12] := 3.8146973e-06, [44] := 50.0, [47] := 15.0, [48] := 25.0, [49] := 2.0, [51] := 15.0, [52] := 440.0, [54] := 20.0, [55] := 25.0, [56] := 40.0, [57] := 110.0, [58] := -0.25, [59] := 15.0, [60] := 20.0, [67] := 225.0, [68] := 15.0, [72] := 197.40001);
   p12_recirc_input_max : REAL := 1750.0;
   p12_recirc_input_min : REAL;
   p12_recirc_output_max : REAL := 1750.0;
   p12_recirc_output_min : REAL;
   p12r01 : routine := (comment := 7);
   p12r02 : routine := (comment := -1073741761);
   p12r02_fault_exists : BOOL;
   p12r02_not_safe_temp : BOOL := 1;
   p12r02_safe_temp : BOOL;
   p12r02_shutdown_temp : BOOL;
   p12r02_timer_fault : TIMER[4];
   p12r02_timer_safe_temp : TIMER[2] := ([0].PRE := 30000, [1].PRE := 30000, [1].ACC := 30015, [1].EN := 1, [1].DN := 1);
   p12r02_timer_warning : TIMER[4] := ([0].PRE := 1500);
   p12r02_unack_fault : BOOL;
   p12r02_unack_warning : BOOL := 1;
   p12r02_warning_exists : BOOL := 1;
   p12r03 : routine := (comment := -1073741761);
   p12r03_hz : SYS_SCP := (Input_Max := 1750.0, Output_Max := 60.0, Output := 3.8146973e-06);
   p12r03_timer_fault : TIMER[4];
   p12r03_timer_warning : TIMER[4];
   p12r04 : routine := (comment := -1073741761);
   p12r04_timer_fault : TIMER[4];
   p12r04_timer_warning : TIMER[4];
   p12r05 : routine := (comment := -1073741761);
   p12r05_exh_status : DINT := 3;
   p12r05_recirc_status : DINT := 3;
   p12r05_Temp_ctl_status : DINT := 4;
   p12r05_timer_fault : TIMER[4];
   p12r05_timer_warning : TIMER[4];
   p12r06 : routine := (comment := -1073741572);
   p12r06_timer_fault : TIMER[4];
   p12r06_timer_warning : TIMER[4];
   p12r07 : routine := (comment := -1073741761);
   p12r07_timer_fault : TIMER[4];
   p12r07_timer_warning : TIMER[4];
   p12r08 : routine := (comment := -1073741761);
   p12r08_timer_fault : TIMER[4];
   p12r08_timer_warning : TIMER[4];
   p12r09 : routine := (comment := -1073741761);
   p12r09_timer_fault : TIMER[4];
   p12r09_timer_warning : TIMER[8];
   p12r10 : routine := (comment := -1073741761);
   p12r10_timer_fault : TIMER[4];
   p12r10_timer_warning : TIMER[4];
   p12r15_mtr_roll_speed_offset : REAL;
   p12r16_pid_temp_cv : DINT;
   p12r16_temp_ok : BOOL := 1;
   p12r20 : routine := (comment := -1073741761);
   p12r20_safeties_ok : BOOL;
   p12r20_state : DINT := 5;
   p12r20_status : DINT := 2;
   p12r20_timer_fault : TIMER[4];
   p12r20_timer_state_11 : TIMER := (PRE := 5000, ACC := 5020, EN := 1, DN := 1);
   p12r20_timer_state_3 : TIMER := (PRE := 1000);
   p12r20_timer_state_4 : TIMER := (PRE := 1000);
   p12r20_timer_state_7 : TIMER := (PRE := 2000);
   p12r20_timer_warning : TIMER[4];
   p12r30 : routine := (comment := -1073741697, warning := 128, warning_ack := 128);
   p12r30_cv_man_sp : REAL := 15.0;
   p12r30_pb_auto : BOOL;
   p12r30_pb_manual : BOOL;
   p12r30_pb_zone_off : BOOL;
   p12r30_pb_zone_on : BOOL;
   p12r30_permissive_run : BOOL;
   p12r30_pid_temp : PID := (CTL := -2077195136, EN := 1, SWM := 1, NOBC := 1, NOZC := 1, INI := 1, DVNA := 1, PVHA := 1, KP := 25.0, KI := 2.0, BIAS := 15.0, MAXS := 1000.0, MAXO := 100.0, UPD := 0.01, PV := 196.7, ERR := -196.7, MAXI := 10000.0, MAXCV := 100.0, MAXTIE := 4095.0, DATA[0] := 476.75, DATA[1] := -314.72, DATA[2] := 196.7, DATA[3] := -196.7, DATA[5] := 0.1, DATA[6] := 0.1, DATA[7] := 0.16, DATA[8] := 25.0, DATA[9] := 2.0, DATA[11] := 25.0, DATA[12] := 2.0, DATA[15] := 1.0, DATA[16] := 0.024420025);
   p12r30_pid_temp_pv : REAL := 1974.0001;
   p12r30_pid_temp_sp : REAL := 225.0;
   p12r30_pid_temp_sp_error : REAL := 197.40001;
   p12r30_pid_temp_sp_last : REAL := 225.0;
   p12r30_request_deviation_warning : BOOL;
   p12r30_request_heat : BOOL;
   p12r30_request_heat_last : BOOL;
   p12r30_request_manual : BOOL;
   p12r30_request_PID_shot : BOOL;
   p12r30_request_soak_control : BOOL := 1;
   p12r30_temp_deviation_setpoint : DINT := 5;
   p12r30_timer_fault : TIMER[16] := ([0].PRE := 5000, [2].PRE := 1000, [4].PRE := 1000, [10].PRE := 5000, [11].PRE := 5000, [12].PRE := 5000);
   p12r30_timer_warning : TIMER[12] := ([0].PRE := 10000, [1].PRE := 1000, [2].PRE := 1000, [3].PRE := 90000, [4].PRE := 1000, [6].PRE := 1000, [7].PRE := 1000, [7].ACC := 1010, [7].EN := 1, [7].DN := 1, [8].PRE := 1000);
   p12r30_vfds_ok : BOOL;
   p12r30_vfds_ready : BOOL := 1;
   p12r31 : routine := (comment := -1073741697, warning := 1, unack_warning := 1);
   p12r31_pb_start : BOOL;
   p12r31_pb_stop : BOOL;
   p12r31_request_auto_run : BOOL;
   p12r31_request_auto_stop : BOOL := 1;
   p12r31_run_permissive : BOOL := 1;
   p12r31_timer_fault : TIMER[5] := ([1].PRE := 500);
   p12r31_timer_warning : TIMER[5] := ([0].PRE := 10000, [0].ACC := 10014, [0].EN := 1, [0].DN := 1, [1].PRE := 20000, [2].PRE := 500);
   p12r31_vfd_stopped : BOOL := 1;
   p12r32 : routine := (comment := -536870849, warning := 1, unack_warning := 1);
   p12r32_fan_pb_stopped : BOOL;
   p12r32_pb_start : BOOL;
   p12r32_pb_stop : BOOL;
   p12r32_request_auto_run : BOOL;
   p12r32_request_auto_stop : BOOL := 1;
   p12r32_run_permissive : BOOL := 1;
   p12r32_timer_fault : TIMER[5] := ([1].PRE := 500);
   p12r32_timer_warning : TIMER[5] := ([0].PRE := 10000, [0].ACC := 10014, [0].EN := 1, [0].DN := 1, [1].PRE := 20000, [2].PRE := 20000);
   p12r32_vfd_stopped : BOOL := 1;
   p13_ai_exhaust_amps : REAL;
   p13_ai_exhaust_hz : REAL := 3.8146973e-06;
   p13_ai_exhaust_hz_max : REAL := 60.0;
   p13_ai_exhaust_pct : REAL;
   p13_ai_exhaust_rpm : REAL;
   p13_ai_recirc_amps : REAL;
   p13_ai_recirc_hz : REAL := 3.8146973e-06;
   p13_ai_recirc_hz_max : REAL := 60.0;
   p13_ai_recirc_pct : REAL;
   p13_ai_recirc_rpm : REAL;
   p13_ai_tc01 : REAL := 66.5;
   p13_ai_tc02 : REAL := 65.6;
   p13_ao_cv : REAL;
   p13_ao_exhaust_selected_speed : REAL;
   p13_ao_recirc_selected_speed : REAL;
   p13_di_door_open : BOOL;
   p13_di_exh : acs800_di_normal := (ready := 1, ctrl_from_net := 1, ref_from_net := 1);
   p13_di_exh_fan_mtr_ts : BOOL := 1;
   p13_di_exh_flow_ok : BOOL;
   p13_di_filter_clean : BOOL := 1;
   p13_di_recirc : acs800_di_normal := (ready := 1, ctrl_from_net := 1, ref_from_net := 1);
   p13_di_recirc_fan_mtr_ts : BOOL := 1;
   p13_di_recirc_flow_ok : BOOL;
   p13_di_tc01_bo : BOOL;
   p13_di_tc02_bo : BOOL;
   p13_dint_to_hmi : DINT[16] := ([4] := 655971, [5] := 1060, [6] := 28784, [8] := 1, [9] := 1, [10] := 3, [11] := 3);
   p13_do_exh : acs800_do_normal;
   p13_do_recirc : acs800_do_normal;
   p13_exhaust_input_max : REAL := 2000.0;
   p13_exhaust_input_min : REAL;
   p13_exhaust_output_max : REAL := 2000.0;
   p13_exhaust_output_min : REAL;
   p13_hc_input_max : REAL := 100.0;
   p13_hc_input_min : REAL;
   p13_hc_output_max : REAL := 30840.0;
   p13_hc_output_min : REAL;
   p13_param_fast_to_soak : REAL := 5.0;
   p13_param_lfl_hhl : REAL := 40.0;
   p13_param_lfl_hl : REAL := 25.0;
   p13_param_pid1_ff : REAL;
   p13_param_pid1_kd : REAL;
   p13_param_pid1_ki : REAL := 0.1;
   p13_param_pid1_kp : REAL := 10.0;
   p13_param_pid2_ff : REAL;
   p13_param_pid2_kd : REAL;
   p13_param_pid2_ki : REAL := 0.22;
   p13_param_pid2_kp : REAL := 75.0;
   p13_param_shutdown_temp : REAL := 125.0;
   p13_param_soak_to_fast : REAL := 15.0;
   p13_param_tc01_dev : REAL := 25.0;
   p13_param_tc01_hl : REAL := 400.0;
   p13_param_tc01z : REAL;
   p13_param_tc02z : REAL;
   p13_param_zone_pressure : REAL;
   p13_real_to_hmi : REAL[112] := ([0] := 66.9, [1] := 66.0, [2] := 66.9, [8] := 3.8146973e-06, [12] := 3.8146973e-06, [44] := 10.0, [45] := 0.1, [48] := 75.0, [49] := 0.22, [52] := 400.0, [54] := 25.0, [55] := 25.0, [56] := 40.0, [57] := 125.0, [59] := 5.0, [60] := 15.0, [67] := 70.0, [68] := 100.0, [72] := 66.9);
   p13_recirc_input_max : REAL := 2000.0;
   p13_recirc_input_min : REAL;
   p13_recirc_output_max : REAL := 2000.0;
   p13_recirc_output_min : REAL;
   p13r01 : routine := (comment := 7);
   p13r02 : routine := (comment := -1073741761);
   p13r02_fault_exists : BOOL;
   p13r02_not_safe_temp : BOOL;
   p13r02_safe_temp : BOOL := 1;
   p13r02_shutdown_temp : BOOL := 1;
   p13r02_timer_fault : TIMER[4];
   p13r02_timer_safe_temp : TIMER[2] := ([0].PRE := 30000, [0].ACC := 30016, [0].EN := 1, [0].DN := 1, [1].PRE := 30000);
   p13r02_timer_warning : TIMER[4] := ([0].PRE := 1500);
   p13r02_unack_fault : BOOL;
   p13r02_unack_warning : BOOL;
   p13r02_warning_exists : BOOL;
   p13r03 : routine := (comment := -1073741761);
   p13r03_hz : SYS_SCP := (Input_Max := 1800.0, Output_Max := 60.0, Output := -3.8146973e-06);
   p13r03_timer_fault : TIMER[4];
   p13r03_timer_warning : TIMER[4];
   p13r04 : routine := (comment := -1073741761);
   p13r04_timer_fault : TIMER[4];
   p13r04_timer_warning : TIMER[4];
   p13r05 : routine := (comment := -1073741761);
   p13r05_exh_status : DINT := 3;
   p13r05_recirc_status : DINT := 3;
   p13r05_temp_ctl_status : DINT := 1;
   p13r05_timer_fault : TIMER[4];
   p13r05_timer_warning : TIMER[4];
   p13r06 : routine := (comment := -1073741572);
   p13r06_timer_fault : TIMER[4];
   p13r06_timer_warning : TIMER[4];
   p13r07 : routine := (comment := -1073741761);
   p13r07_timer_fault : TIMER[4];
   p13r07_timer_warning : TIMER[4];
   p13r08 : routine := (comment := -1073741761);
   p13r08_timer_fault : TIMER[4];
   p13r08_timer_warning : TIMER[4];
   p13r09 : routine := (comment := -1073741761);
   p13r09_timer_fault : TIMER[4];
   p13r09_timer_warning : TIMER[8];
   p13r10 : routine := (comment := -1073741761);
   p13r10_timer_fault : TIMER[4];
   p13r10_timer_warning : TIMER[4];
   p13r16_pid_temp_cv : DINT;
   p13r20 : routine := (comment := -1073741761);
   p13r20_state : DINT := 3;
   p13r20_status : DINT := 1;
   p13r20_timer_fault : TIMER[4];
   p13r20_timer_state_11 : TIMER := (PRE := 5000, ACC := 5001);
   p13r20_timer_state_3 : TIMER := (PRE := 1000);
   p13r20_timer_state_4 : TIMER := (PRE := 1000);
   p13r20_timer_state_7 : TIMER := (PRE := 2000);
   p13r20_timer_warning : TIMER[4];
   p13r30 : routine := (comment := -1073741697);
   p13r30_cv_man_sp : REAL := 100.0;
   p13r30_pb_auto : BOOL;
   p13r30_pb_manual : BOOL;
   p13r30_pb_zone_off : BOOL;
   p13r30_pb_zone_on : BOOL;
   p13r30_permissive_run : BOOL := 1;
   p13r30_pid_temp_pv : REAL := 66.5;
   p13r30_pid_temp_sp : REAL := 70.0;
   p13r30_pid_temp_sp_error : REAL := 32.6;
   p13r30_pid_temp_sp_last : REAL := 70.0;
   p13r30_request_cool : BOOL;
   p13r30_request_deviation_warning : BOOL;
   p13r30_request_manual : BOOL;
   p13r30_request_PID_shot : BOOL;
   p13r30_temp_deviation_setpoint : DINT := 5;
   p13r30_temp_pid_ctrl : PID := (CTL := -2043640704, EN := 1, SWM := 1, CA := 1, NOBC := 1, NOZC := 1, INI := 1, DVNA := 1, PVHA := 1, SP := 100.0, KP := 75.0, KI := 0.22, MAXS := 1000.0, MAXO := 100.0, UPD := 0.1, PV := 66.200005, ERR := -33.799995, MAXI := 1000.0, MAXCV := 100.0, MAXTIE := 4095.0, DATA[0] := 253.49997, DATA[1] := 105.920006, DATA[2] := 66.200005, DATA[3] := -33.799995, DATA[4] := 100.0, DATA[5] := 0.1, DATA[6] := 1.0, DATA[7] := 1.6, DATA[8] := 75.0, DATA[9] := 0.22, DATA[11] := 75.0, DATA[12] := 0.22, DATA[15] := 1.0, DATA[16] := 0.024420025);
   p13r30_timer_fault : TIMER[16] := ([0].PRE := 5000, [2].PRE := 1000, [4].PRE := 1000);
   p13r30_timer_warning : TIMER[12] := ([0].PRE := 10000, [1].PRE := 1000, [2].PRE := 1000, [3].PRE := 90000, [4].PRE := 1000, [5].PRE := 90000, [6].PRE := 1000, [7].PRE := 1000, [8].PRE := 1000);
   p13r30_vfds_ready : BOOL := 1;
   p13r31 : routine := (comment := -1073741697);
   p13r31_pb_start : BOOL;
   p13r31_pb_stop : BOOL;
   p13r31_request_auto_run : BOOL;
   p13r31_request_auto_stop : BOOL := 1;
   p13r31_run_permissive : BOOL := 1;
   p13r31_timer_fault : TIMER[5] := ([1].PRE := 500);
   p13r31_timer_warning : TIMER[5] := ([0].PRE := 10000, [1].PRE := 20000, [2].PRE := 500);
   p13r31_vfd_stopped : BOOL := 1;
   p13r32 : routine := (comment := -536870849);
   p13r32_pb_start : BOOL;
   p13r32_pb_stop : BOOL;
   p13r32_request_auto_run : BOOL;
   p13r32_request_auto_stop : BOOL;
   p13r32_run_permissive : BOOL := 1;
   p13r32_timer_fault : TIMER[5] := ([1].PRE := 500);
   p13r32_timer_warning : TIMER[5] := ([0].PRE := 10000, [1].PRE := 20000, [2].PRE := 20000);
   p13r32_vfd_stopped : BOOL := 1;
   p19_ai_prs : REAL := 15.128405;
   p19_ai_tc01 : REAL := 65.4;
   p19_ao_cv : REAL;
   p19_di_pump : BOOL;
   p19_di_tc01_bo : BOOL;
   p19_di_tc02_bo : BOOL := 1;
   p19_dint_to_hmi : DINT[16] := ([0] := 655360, [1] := 32768, [5] := 16382);
   p19_do_pump : BOOL;
   p19_flow_input_max : REAL := 100.0;
   p19_flow_input_min : REAL;
   p19_flow_output_max : REAL := 30840.0;
   p19_flow_output_min : REAL;
   p19_param_pid1_ff : REAL;
   p19_param_pid1_kd : REAL;
   p19_param_pid1_ki : REAL;
   p19_param_pid1_kp : REAL;
   p19_param_pid2_ff : REAL;
   p19_param_pid2_kd : REAL;
   p19_param_pid2_ki : REAL := 1.0;
   p19_param_pid2_kp : REAL := 50.0;
   p19_param_prs_offset : REAL := 6.0;
   p19_param_tc01_dev : REAL := 20.0;
   p19_param_tc01z : REAL;
   p19_param_tc02z : REAL;
   p19_param_zone_pressure : REAL := 10.0;
   p19_prs_input_max : REAL := 100.0;
   p19_prs_input_min : REAL;
   p19_prs_output_max : REAL := 30840.0;
   p19_prs_output_min : REAL;
   p19_real_to_hmi : REAL[80] := ([0] := 65.6, [1] := 2192.0, [2] := 65.6, [6] := 14.7393, [48] := 50.0, [49] := 1.0, [54] := 20.0, [58] := 10.0, [68] := 100.0, [72] := 65.6);
   p19r01 : routine := (comment := 7);
   p19r02 : routine := (comment := -1073741761);
   p19r02_fault_exists : BOOL;
   p19r02_timer_fault : TIMER[4];
   p19r02_timer_warning : TIMER[4] := ([0].PRE := 1500);
   p19r02_unack_fault : BOOL;
   p19r02_unack_warning : BOOL;
   p19r02_warning_exists : BOOL;
   p19r03 : routine := (comment := -1073741761);
   p19r03_flow_scp : SYS_SCP := (Input_Max := 100.0, Output_Max := 30840.0);
   p19r03_prs_input_max : REAL := 30840.0;
   p19r03_prs_input_min : REAL;
   p19r03_prs_output_max : REAL := 50.0;
   p19r03_prs_output_min : REAL;
   p19r03_prs_scp : SYS_SCP := (Input := 60.0, Input_Max := 100.0, Output_Max := 30840.0, Output := 18504.0);
   p19r03_timer_fault : TIMER[4];
   p19r03_timer_warning : TIMER[4];
   p19r04 : routine := (comment := -1073741761);
   p19r04_timer_fault : TIMER[4];
   p19r04_timer_warning : TIMER[4];
   p19r05 : routine := (comment := -1073741761);
   p19r05_timer_fault : TIMER[4];
   p19r05_timer_warning : TIMER[4];
   p19r06 : routine := (comment := -1073741572);
   p19r06_timer_fault : TIMER[4];
   p19r06_timer_warning : TIMER[4];
   p19r07 : routine := (comment := -1073741761);
   p19r07_timer_fault : TIMER[4];
   p19r07_timer_warning : TIMER[4];
   p19r08 : routine := (comment := -1073741761);
   p19r08_timer_fault : TIMER[4];
   p19r08_timer_warning : TIMER[4];
   p19r09 : routine := (comment := -1073741761);
   p19r09_timer_fault : TIMER[4];
   p19r09_timer_warning : TIMER[4];
   p19r10 : routine := (comment := -1073741761);
   p19r10_timer_fault : TIMER[4];
   p19r10_timer_warning : TIMER[4];
   p19r16_pid_temp_cv : DINT;
   p19r30 : routine := (comment := -1073741697);
   p19r30_cv_man_sp : REAL := 100.0;
   p19r30_pb_auto : BOOL;
   p19r30_pb_manual : BOOL;
   p19r30_pb_zone_off : BOOL;
   p19r30_pb_zone_on : BOOL;
   p19r30_permissive_run : BOOL := 1;
   p19r30_pid_temp : PID := (CTL := -2110741376, EN := 1, CA := 1, NOBC := 1, NOZC := 1, INI := 1, OLL := 1, DVNA := 1, PVHA := 1, SP := 100.0, KP := 50.0, KI := 1.0, MAXS := 1000.0, MAXO := 100.0, UPD := 0.01, PV := 65.1, ERR := -34.9, MAXI := 10000.0, MAXCV := 100.0, MAXTIE := 4095.0, DATA[0] := 23.445763, DATA[1] := 104.159996, DATA[2] := 65.1, DATA[3] := -34.9, DATA[4] := 100.0, DATA[5] := 0.1, DATA[6] := 0.1, DATA[7] := 0.16, DATA[8] := 50.0, DATA[9] := 1.0, DATA[11] := 50.0, DATA[12] := 1.0, DATA[15] := 1.0, DATA[16] := 0.024420025);
   p19r30_pid_temp_pv : DINT := 653;
   p19r30_pid_temp_sp : DINT := 65;
   p19r30_request_cool : BOOL;
   p19r30_request_manual : BOOL;
   p19r30_timer_fault : TIMER[4] := ([2].PRE := 1000);
   p19r30_timer_warning : TIMER[4] := ([0].PRE := 10000, [1].PRE := 1000, [2].PRE := 1000, [2].ACC := 1007, [2].EN := 1, [2].DN := 1, [3].PRE := 90000);
   p19r31 : routine := (comment := -1073741761);
   p19r31_pb_start : BOOL;
   p19r31_pb_stop : BOOL;
   p19r31_request_a00 : BOOL;
   p19r31_request_auto_run : BOOL;
   p19r31_request_manual_run : BOOL;
   p19r31_run_permissive : BOOL := 1;
   p19r31_timer_fault : TIMER[4] := ([0].PRE := 5000, [1].PRE := 2000, [2].ACC := 3);
   p19r31_timer_warning : TIMER[4];
   p20_acc_ctr_prs_input_max : REAL := 100.0;
   p20_acc_ctr_prs_input_min : REAL;
   p20_acc_ctr_prs_output_max : REAL := 30840.0;
   p20_acc_ctr_prs_output_min : REAL;
   p20_acc_fill_prs : REAL := 90.0;
   p20_acc_fill_prs_input_max : REAL := 100.0;
   p20_acc_fill_prs_input_min : REAL;
   p20_acc_fill_prs_output_max : REAL := 30840.0;
   p20_acc_fill_prs_output_min : REAL;
   p20_acc_fill_time_sec : REAL;
   p20_acc_input_max : REAL := 7496.0;
   p20_acc_input_min : REAL := 22420.0;
   p20_acc_output_max : REAL := 40.0;
   p20_acc_output_min : REAL;
   p20_acc_ten_prs_input_max : REAL := 100.0;
   p20_acc_ten_prs_input_min : REAL;
   p20_acc_ten_prs_output_max : REAL := 30840.0;
   p20_acc_ten_prs_output_min : REAL;
   p20_acc_tens_prs : REAL := 57.08;
   p20_ai_acc_pstn : REAL := 0.053604126;
   p20_ai_lc01 : REAL := 0.9266419;
   p20_ai_letoff_dia : REAL := 23.59639;
   p20_ai_lo_turret_amps : REAL;
   p20_ai_lo_turret_hz : REAL := -3.8146973e-06;
   p20_ai_lo_turret_speed : REAL;
   p20_ai_loa_speed : REAL;
   p20_ai_lob_speed : REAL;
   p20_ao_acc_ctr_prs : REAL := 10.0;
   p20_ao_acc_fill_prs : REAL := 32.0;
   p20_ao_acc_ten_prs : REAL := 32.0;
   p20_ao_lo_turret_selected_speed : REAL;
   p20_ao_loa_selected_speed : REAL;
   p20_ao_loa_torque : REAL := 300.0;
   p20_ao_lob_selected_speed : REAL;
   p20_ao_lob_torque : REAL := 300.0;
   p20_di_acc_door_open : BOOL;
   p20_di_acc_empty : BOOL := 1;
   p20_di_acc_full : BOOL;
   p20_di_clutch_prs_ok : BOOL;
   p20_di_lfr_jog_fwd : BOOL;
   p20_di_lfr_jog_rev : BOOL;
   p20_di_lfr_nip_close : BOOL;
   p20_di_lo_turret : acs800_di_normal := (ready := 1, ctrl_from_net := 1, ref_from_net := 1);
   p20_di_lo_turret_therm : BOOL := 1;
   p20_di_loa_active : BOOL;
   p20_di_loa_brake : BOOL := 1;
   p20_di_loa_fwd_dir : BOOL := 1;
   p20_di_loa_jog : BOOL;
   p20_di_loa_start : BOOL;
   p20_di_loa_stop : BOOL := 1;
   p20_di_loa_temp : BOOL := 1;
   p20_di_lob_brake_thermostat : BOOL := 1;
   p20_di_lob_fwd_dir : BOOL := 1;
   p20_di_lob_jog : BOOL;
   p20_di_lob_motor_thermostat : BOOL := 1;
   p20_di_lob_start : BOOL;
   p20_di_lob_stop : BOOL := 1;
   p20_di_lof_acc_fill : BOOL;
   p20_di_turret_fwd : BOOL;
   p20_di_turret_pos : BOOL := 1;
   p20_di_turret_rev : BOOL;
   p20_dia_input_max : REAL := 30959.0;
   p20_dia_input_min : REAL := 100.0;
   p20_dia_output_max : REAL := 55.0;
   p20_dia_output_min : REAL := 4.0;
   p20_dint_to_hmi : DINT[16] := ([0] := 38, [1] := 7368816, [2] := 320, [4] := 48, [6] := 131072, [7] := 1);
   p20_do_acc_enable_tension : BOOL := 1;
   p20_do_acc_high_prs : BOOL;
   p20_do_close_nip : BOOL;
   p20_do_enable_lfr_fwd : BOOL;
   p20_do_enable_lfr_rev : BOOL;
   p20_do_engage_lfr_clutch : BOOL;
   p20_do_wdr_turret : acs800_do_normal;
   p20_lc_input_max : REAL := 10000.0;
   p20_lc_input_min : REAL;
   p20_lc_output_max : REAL := 250.0;
   p20_lc_output_min : REAL;
   p20_loa_ai_amps : REAL;
   p20_loa_ai_hz : REAL := 3.8146973e-06;
   p20_loa_ai_rpm : REAL;
   p20_loa_ai_torque : REAL;
   p20_loa_footage_input_max : REAL := 9000.0;
   p20_loa_footage_input_min : REAL;
   p20_loa_footage_output_max : REAL := 990.0;
   p20_loa_footage_output_min : REAL;
   p20_lob_ai_amps : REAL;
   p20_lob_ai_hz : REAL := -3.8146973e-06;
   p20_lob_ai_rpm : REAL;
   p20_lob_ai_torque : REAL := 17.4;
   p20_lob_footage_input_max : REAL := 9000.0;
   p20_lob_footage_input_min : REAL;
   p20_lob_footage_output_max : REAL := 1000.0;
   p20_lob_footage_output_min : REAL;
   p20_param_acc_auto_fill : REAL := 10.0;
   p20_param_acc_ctr_prs : REAL := 10.0;
   p20_param_acc_empty_prs : REAL := 32.0;
   p20_param_acc_fast_accel : REAL := 100.0;
   p20_param_acc_fast_decel : REAL := 100.0;
   p20_param_acc_fill_ctr_prs : REAL := 10.0;
   p20_param_acc_high_prs : REAL := 10.0;
   p20_param_acc_init_high_prs : REAL := 3.5;
   p20_param_acc_init_low_prs : REAL := 3.0;
   p20_param_acc_init_prs : REAL := 3.0;
   p20_param_acc_med_accel : REAL := 1.0;
   p20_param_acc_med_decel : REAL := 1.0;
   p20_param_acc_pid_accel : REAL := 2.0;
   p20_param_acc_pid_decel : REAL := 2.0;
   p20_param_acc_pos_prs : REAL := 10.0;
   p20_param_acc_slow_accel : REAL := 0.5;
   p20_param_acc_slow_decel : REAL := 0.5;
   p20_param_empty_pct : REAL := 0.5;
   p20_param_high_accel_rate : REAL := 100.0;
   p20_param_high_ctrl_pct : REAL := 60.0;
   p20_param_high_decel_rate : REAL := 100.0;
   p20_param_high_ki : REAL := 0.01;
   p20_param_high_kp : REAL := 1000.0;
   p20_param_high_low_ctrl_pct : REAL := 10.0;
   p20_param_high_upd : REAL := 0.01;
   p20_param_jog_accel_rate : REAL := 10.0;
   p20_param_jog_decel_rate : REAL := 10.0;
   p20_param_letoff_jog_speed : REAL := 20.0;
   p20_param_lo_turret_gear_ratio : REAL := 1200.0;
   p20_param_lo_turret_index_speed : REAL := 8.0;
   p20_param_loa_gear_ratio : REAL := 50.86;
   p20_param_lob_gear_ratio : REAL := 50.86;
   p20_param_lof_fast_fill : REAL := 50.0;
   p20_param_lof_slow_fill : REAL := 40.0;
   p20_param_lof_stop_fill : REAL := 30.0;
   p20_param_low_ctrl_pct : REAL := 7.0;
   p20_param_low_low_ctrl_pct : REAL := 2.0;
   p20_param_norm_accel_rate : REAL := 2.0;
   p20_param_norm_decel_rate : REAL := 20.0;
   p20_param_prs_accel_rate : REAL := 1.0;
   p20_param_prs_decel_rate : REAL := 1.0;
   p20_param_run_torque : REAL := 300.0;
   p20_real_to_hmi : REAL[112] := ([0] := 0.95815134, [1] := 23.56334, [2] := 0.18760681, [8] := 3.8146973e-06, [14] := -3.8146973e-06, [15] := 65.0, [20] := -3.8146973e-06, [22] := 17.5727, [25] := 10.0, [26] := 32.0, [27] := 32.0, [40] := 1.8, [41] := 2.0);
   p20_request_run_index_dir : BOOL;
   p20_request_run_index_rev_dir : BOOL;
   p20_vfd_di_loa : acs800_di_normal := (ready := 1, ctrl_from_net := 1, ref_from_net := 1);
   p20_vfd_di_lob : acs800_di_normal := (ready := 1, ctrl_from_net := 1, ref_from_net := 1);
   p20_vfd_do_loa : acs800_do_normal;
   p20_vfd_do_lob : acs800_do_normal;
   p20_zero_tension_prs : REAL := 38.0;
   p20r01 : routine := (comment := 7);
   p20r02 : routine := (comment := -1073741761, oneshot := 1);
   p20r02_fault_exists : BOOL := 1;
   p20r02_letoff_dia_ft : REAL := 1.9720192;
   p20r02_letoff_selection_dwell : TIMER := (PRE := 60000, ACC := 60000);
   p20r02_timer_fault : TIMER[4];
   p20r02_timer_warning : TIMER[4];
   p20r02_unack_fault : BOOL := 1;
   p20r02_unack_warning : BOOL := 1;
   p20r02_warning_exists : BOOL := 1;
   p20r03 : routine := (comment := -1073741761);
   p20r03_accumulator_pct_scp : SYS_SCP := (Input := 22392.0, Input_Min := 22420.0, Input_Max := 7496.0, Output_Max := 100.0, Output := 0.18760681);
   p20r03_accumulator_scp : SYS_SCP := (Input := 22392.0, Input_Min := 22420.0, Input_Max := 7496.0, Output_Max := 40.0, Output := 0.07504654);
   p20r03_distance_to_core : REAL := 46.5;
   p20r03_lo_radius : REAL := 11.81472;
   p20r03_lo_turret_speed_fb : SYS_RPM_TO_SPEED := (IN_gear_ratio := 1200.0, IN_roll_diameter := 3.2);
   p20r03_loa_distance_to_core : REAL := 46.52;
   p20r03_Loa_footage_scp : SYS_SCP := (Input := -3.4682617, Input_Max := 9000.0, Output_Max := 990.0);
   p20r03_loa_speed_fb : SYS_RPM_TO_SPEED := (IN_gear_ratio := 50.86, IN_roll_diameter := 1.9720192);
   p20r03_load_cell : SYS_SCP := (Input := 37.85083, Input_Max := 10000.0, Output_Max := 250.0, Output := 0.94627076);
   p20r03_lob_distance_to_core : REAL := 46.5;
   p20r03_Lob_footage_scp : SYS_SCP := (Input := 158.0127, Input_Max := 9000.0, Output_Max := 1000.0, Output := 17.556967);
   p20r03_lob_speed_fb : SYS_RPM_TO_SPEED := (IN_gear_ratio := 50.86, IN_roll_diameter := 1.9720192);
   p20r03_sensor_input : REAL := 34.733208;
   p20r03_sensor_scp : SYS_SCP := (Input := 18687.0, Input_Min := 100.0, Input_Max := 30959.0, Output_Min := 4.0, Output_Max := 55.0, Output := 34.71833);
   p20r03_timer_fault : TIMER[4];
   p20r03_timer_warning : TIMER[4];
   p20r04 : routine := (comment := -1073741761);
   p20r04_acc_ctr_prs : SYS_SCP := (Input := 10.0, Input_Max := 100.0, Output_Max := 30840.0, Output := 3084.0);
   p20r04_acc_fill_prs : SYS_SCP := (Input := 32.0, Input_Max := 100.0, Output_Max := 30840.0, Output := 9868.8);
   p20r04_acc_ten_prs : SYS_SCP := (Input := 32.0, Input_Max := 100.0, Output_Max := 30840.0, Output := 9868.8);
   p20r04_lo_turret_speed_to_vfd : SYS_SPEED_TO_VFD := (IN_gear_ratio := 1200.0, IN_roll_diameter := 3.2);
   p20r04_loa_speed_to_vfd : SYS_SPEED_TO_VFD := (IN_gear_ratio := 50.86, IN_roll_diameter := 1.9720192);
   p20r04_lob_speed_to_vfd : SYS_SPEED_TO_VFD := (IN_gear_ratio := 50.86, IN_roll_diameter := 1.9720192);
   p20r04_timer_fault : TIMER[4];
   p20r04_timer_warning : TIMER[4];
   p20r05 : routine := (comment := -1073741761);
   p20r05_timer_fault : TIMER[4];
   p20r05_timer_warning : TIMER[4];
   p20r06 : routine := (comment := -1073741572);
   p20r06_ave_lc : REAL := 0.9646084;
   p20r06_lc_ave_ctrl : CONTROL := (LEN := 19);
   p20r06_lc_buffer : REAL[20] := ([0] := 1.0051575, [1] := 0.96589965, [2] := 1.0002502, [3] := 0.9560852, [4] := 0.9855286, [5] := 0.97571415, [6] := 0.92173463, [7] := 0.9413635, [8] := 0.90701294, [9] := 1.0051575, [10] := 0.97571415, [11] := 1.0051575, [12] := 0.9708069, [13] := 0.96099246, [14] := 0.951178, [15] := 0.9364563, [16] := 0.995343, [17] := 0.9708069, [18] := 0.97571415, [19] := 0.9364563);
   p20r06_lc_ctrl : CONTROL := (LEN := 20, POS := 20, DN := 1);
   p20r06_sample_timer : TIMER := (PRE := 200, ACC := 123, EN := 1, TT := 1);
   p20r06_timer_fault : TIMER[4];
   p20r06_timer_warning : TIMER[4];
   p20r06_unload : DINT := 1;
   p20r07 : routine := (comment := -1073741761);
   p20r07_timer_fault : TIMER[4];
   p20r07_timer_warning : TIMER[4];
   p20r08 : routine := (comment := -1073741761);
   p20r08_timer_fault : TIMER[4];
   p20r08_timer_warning : TIMER[4];
   p20r09 : routine := (comment := -1073741761, fault := 1, fault_ack := 1);
   p20r09_acc_toggle : SYS_Toggle;
   p20r09_accumulator_auto : BOOL;
   p20r09_letoff_a_active : BOOL;
   p20r09_timer_fault : TIMER[4];
   p20r09_timer_warning : TIMER[4];
   p20r10 : routine := (comment := -1073739969, oneshot := 1);
   p20r10_param_acc_full_psn : REAL := 100.0;
   p20r10_param_fill_gain : REAL := 0.0198;
   p20r10_param_normal_gain : REAL := 0.0198;
   p20r10_param_psn_gain : REAL := 0.0198;
   p20r10_pid_psn : PID := (CTL := -2078244224, EN := 1, SWM := 1, NOBC := 1, INI := 1, DVPA := 1, PVHA := 1, SP := 100.0, KP := 180.0, BIAS := 5.0, MAXS := 100.0, SO := 100.0, MAXO := 100.0, UPD := 0.01, PV := 0.18760681, ERR := 99.81239, OUT := 100.0, MAXI := 100.0, MAXCV := 100.0, MAXTIE := 100.0, DATA[1] := -3.001709, DATA[2] := 0.18760681, DATA[3] := 99.81239, DATA[4] := 100.0, DATA[5] := 1.0, DATA[6] := 1.0, DATA[7] := 0.16, DATA[8] := 180.0, DATA[11] := 180.0, DATA[15] := 1.0, DATA[16] := 1.0);
   p20r10_pid_psn_cv : REAL := 100.0;
   p20r10_pid_psn_pv : REAL := 0.18760681;
   p20r10_pid_tens : PID := (CTL := -2078244224, EN := 1, SWM := 1, NOBC := 1, INI := 1, DVPA := 1, PVHA := 1, SP := 15.0, KP := 1.8, KI := 2.0, MAXS := 500.0, SO := 65.0, MAXO := 100.0, UPD := 0.01, PV := 0.98062134, ERR := 14.019379, OUT := 65.0, MAXI := 500.0, MAXCV := 100.0, MAXTIE := 100.0, DATA[0] := 59.953026, DATA[1] := -3.1379883, DATA[2] := 0.98062134, DATA[3] := 14.019379, DATA[4] := 15.0, DATA[5] := 0.2, DATA[6] := 1.0, DATA[7] := 0.16, DATA[8] := 1.8, DATA[9] := 2.0, DATA[11] := 1.8, DATA[12] := 2.0, DATA[15] := 1.0, DATA[16] := 1.0);
   p20r10_pid_tens_cv : REAL := 65.0;
   p20r10_pid_tens_pv : REAL := 0.94627076;
   p20r10_run_permissive : BOOL := 1;
   p20r10_speed_offset : REAL := 0.99;
   p20r10_speed_offset_psn : REAL := 0.99;
   p20r10_speed_offset_tens : REAL := -0.297;
   p20r10_tension_request : BOOL;
   p20r10_timer : TIMER[2] := ([0].PRE := 10, [0].ACC := 30, [0].EN := 1, [0].DN := 1);
   p20r10_timer_fault : TIMER[4];
   p20r10_timer_warning : TIMER[4];
   p20r11 : routine := (comment := -1073741793);
   p20r11_manual_open_nip : BOOL;
   p20r11_nip_close_dwell : TIMER := (PRE := 1000);
   p20r11_permissive_jog : BOOL;
   p20r11_permissive_run : BOOL;
   p20r11_request_close_nip : BOOL;
   p20r11_request_jog_fwd : BOOL;
   p20r11_request_jog_rev : BOOL;
   p20r11_timer_clutch_off : TIMER := (PRE := 300, ACC := 300);
   p20r11_timer_clutch_on : TIMER := (PRE := 300);
   p20r11_timer_fault : TIMER[4];
   p20r11_timer_warning : TIMER[4];
   p20r13 : routine := (comment := -1073741761, oneshot := 1);
   p20r13_acc_top_pos : REAL := 99.7;
   p20r13_ai_acc_pct : REAL := 0.18760681;
   p20r13_ai_loa_footage_ft : REAL;
   p20r13_ai_lob_footage_ft : REAL := 17.556967;
   p20r13_enc : SYS_ENC := (IN_State := 3, OUT_Status := 1);
   p20r13_ramp_tension_pressure : SYS_ACC_DEC_RAMP := (IN_selected_line_speed := 32.0, IN_param_master_accel_rate := 1.0, IN_param_master_decel_rate := 1.0, IN_last_scan_s := 0.031214);
   p20r13_request_fill : BOOL;
   p20r13_selected_pressure : REAL := 32.0;
   p20r13_state : DINT := 3;
   p20r13_status : DINT := 1;
   p20r13_timer_fault : TIMER[4];
   p20r13_timer_warning : TIMER[4];
   p20r14 : routine := (comment := -1073741761, fault := 1, fault_ack := 1);
   p20r14_acc_request_tension_ctrl : BOOL;
   p20r15 : routine := (comment := -536870793);
   p20r15_loa_accel : REAL := 100.0;
   p20r15_loa_accel_decel_ramp : SYS_ACC_DEC_RAMP := (IN_param_master_accel_rate := 100.0, IN_param_master_decel_rate := 100.0, IN_last_scan_s := 0.029428);
   p20r15_loa_decel : REAL := 100.0;
   p20r15_loa_on : BOOL;
   p20r15_loa_selected_speed : REAL;
   p20r15_permissive_run : BOOL;
   p20r15_request_jog_fwd : BOOL;
   p20r15_request_jog_rev : BOOL;
   p20r15_request_over_speed : BOOL;
   p20r15_request_position : BOOL;
   p20r15_request_stop : BOOL := 1;
   p20r15_request_tension : BOOL;
   p20r15_request_thread_fwd : BOOL;
   p20r15_request_thread_rev : BOOL;
   p20r15_timer_fault : TIMER[10];
   p20r15_timer_warning : TIMER[5];
   p20r15_zero_speed : BOOL := 1;
   p20r16 : routine := (comment := -536870793, fault := 5, unack_fault := 1);
   p20r16_loa_accel_decel_ramp : SYS_ACC_DEC_RAMP := (IN_param_master_accel_rate := 100.0, IN_param_master_decel_rate := 100.0, IN_last_scan_s := 0.029566);
   p20r16_lob_accel : REAL := 100.0;
   p20r16_lob_decel : REAL := 100.0;
   p20r16_lob_on : BOOL;
   p20r16_lob_selected_speed : REAL;
   p20r16_permissive_run : BOOL;
   p20r16_request_jog_fwd : BOOL;
   p20r16_request_jog_rev : BOOL;
   p20r16_request_over_speed : BOOL;
   p20r16_request_position : BOOL;
   p20r16_request_stop : BOOL := 1;
   p20r16_request_tension : BOOL;
   p20r16_request_thread_fwd : BOOL;
   p20r16_request_thread_rev : BOOL;
   p20r16_timer_fault : TIMER[10];
   p20r16_timer_warning : TIMER[4];
   p20r16_zero_speed : BOOL := 1;
   p20r17 : routine := (comment := -1073741777);
   p20r17_ave_control : CONTROL := (LEN := 19);
   p20r17_diameter_clac_active : BOOL;
   p20r17_letoff_avg_diam_inch : REAL := 23.66423;
   p20r17_letoff_diam_avg_stack : REAL[20] := ([0] := 23.66249, [1] := 23.59639, [2] := 23.66249, [3] := 23.66249, [4] := 23.66249, [5] := 23.66249, [6] := 23.66249, [7] := 23.66249, [8] := 23.66249, [9] := 23.66249, [10] := 23.66249, [11] := 23.695549, [12] := 23.66249, [13] := 23.695549, [14] := 23.695549, [15] := 23.695549, [16] := 23.66249, [17] := 23.66249, [18] := 23.66249);
   p20r17_stack_ctrl : CONTROL := (LEN := 20, POS := 19);
   p20r17_timer : TIMER[5] := ([0].PRE := 400, [1].PRE := 200);
   p20r17_timer_fault : TIMER[5];
   p20r17_timer_warning : TIMER[5];
   p20r17_winder_a_unload : REAL := 23.62944;
   p20r18 : routine := (comment := -1073741321, warning := 4, unack_warning := 1, state := 3);
   p20r18_acc_dec_ramp : SYS_ACC_DEC_RAMP := (IN_param_master_accel_rate := 8.0, IN_param_master_decel_rate := 8.0, IN_last_scan_s := 0.029438);
   p20r18_accel_rate : REAL := 8.0;
   p20r18_decel_rate : REAL := 8.0;
   p20r18_index_complete : BOOL := 1;
   p20r18_index_move_timer : TIMER := (PRE := 6893);
   p20r18_index_time : DINT := 6893;
   p20r18_index_time_offset : DINT := 1250;
   p20r18_index_timer : TIMER := (PRE := 999999);
   p20r18_pb_index_fwd : BOOL;
   p20r18_pb_index_rev : BOOL;
   p20r18_permissive : BOOL;
   p20r18_request_index_fwd : BOOL;
   p20r18_request_index_rev : BOOL;
   p20r18_selected_speed : REAL;
   p20r18_timer_fault : TIMER[10] := ([3].PRE := 1000);
   p20r18_timer_warning : TIMER[4] := ([1].PRE := 2000, [2].PRE := 2000, [2].ACC := 2022, [2].EN := 1, [2].DN := 1);
   p20r18_zero_speed : BOOL := 1;
   p21_ai_splice_platen_temp : REAL := 367.5;
   p21_ao_splice_platen_temp_cv : REAL;
   p21_di_close_exit_clamp : BOOL;
   p21_di_close_inlet_clamp : BOOL;
   p21_di_open_splice_platen : BOOL;
   p21_di_platen_hi_temp_ok : BOOL := 1;
   p21_di_platen_not_closed : BOOL := 1;
   p21_di_splice_2_hand_close : BOOL;
   p21_di_tc_bo : BOOL;
   p21_dint_to_hmi : DINT[16] := ([10] := 2);
   p21_do_close_exit_clamp_sv : BOOL;
   p21_do_close_inlet_clamp_sv : BOOL;
   p21_do_close_platen_sv : BOOL;
   p21_do_enable_platen_heater : BOOL;
   p21_pid_splice_press_temp : PID := (CTL := -2077195136, EN := 1, SWM := 1, NOBC := 1, NOZC := 1, INI := 1, DVNA := 1, PVHA := 1, KP := 30.0, BIAS := 30.0, MAXS := 1000.0, MAXO := 100.0, UPD := 0.01, PV := 365.9, ERR := -365.9, MAXI := 1000.0, MAXCV := 100.0, MAXTIE := 100.0, DATA[1] := -585.44, DATA[2] := 365.9, DATA[3] := -365.9, DATA[5] := 0.1, DATA[6] := 1.0, DATA[7] := 0.16, DATA[8] := 30.0, DATA[11] := 30.0, DATA[15] := 1.0, DATA[16] := 1.0);
   p21_real_to_hmi : REAL[112] := ([0] := 370.7, [1] := 55.0);
   p21_splice_press_temp_out : SYS_SCP := (Input_Max := 100.0, Output_Max := 32767.0, Output := -0.001953125);
   p21_splice_temp_in_max : REAL := 100.0;
   p21_splice_temp_in_min : REAL;
   p21_splice_temp_out_max : REAL := 32767.0;
   p21_splice_temp_out_min : REAL;
   P21r01 : routine := (comment := 7);
   p21r02 : routine := (comment := -1073741761);
   p21r02_fault_exists : BOOL;
   p21r02_timer_fault : TIMER[4];
   p21r02_timer_warning : TIMER[4];
   p21r02_unack_fault : BOOL;
   p21r02_unack_warning : BOOL;
   p21r02_warning_exists : BOOL;
   p21r03 : routine := (comment := -1073741761);
   p21r03_timer_fault : TIMER[4];
   p21r03_timer_warning : TIMER[4];
   p21r04 : routine := (comment := -1073741761);
   p21r04_timer_fault : TIMER[4];
   p21r04_timer_warning : TIMER[4];
   p21r05 : routine := (comment := -1073741761);
   p21r05_timer_fault : TIMER[4];
   p21r05_timer_warning : TIMER[4];
   p21r06 : routine := (comment := -1073741796);
   p21r06_timer_fault : TIMER[4];
   p21r06_timer_warning : TIMER[4];
   p21r07 : routine := (comment := -1073741761);
   p21r07_timer_fault : TIMER[4];
   p21r07_timer_warning : TIMER[4];
   p21r08 : routine := (comment := -1073741761);
   p21r08_timer_fault : TIMER[4];
   p21r08_timer_warning : TIMER[4];
   p21r09 : routine := (comment := -1073741761);
   p21r09_timer_fault : TIMER[4];
   p21r09_timer_warning : TIMER[4];
   p21r10 : routine := (comment := -1073741761);
   p21r10_index_kd : REAL;
   p21r10_index_ki : REAL := 0.1;
   p21r10_index_kp : REAL := 2.0;
   p21r10_permissive_run : BOOL := 1;
   p21r10_remaining_cure_time : DINT := 55000;
   p21r10_remaining_cure_time_sec : REAL := 55.0;
   p21r10_splice_press_1 : SYS_ENC := (IN_State := 5, OUT_Status := 2);
   p21r10_state : DINT := 5;
   p21r10_status : DINT := 2;
   p21r10_timer_exit_open_delay : TIMER;
   p21r10_timer_fault : TIMER[4];
   p21r10_timer_inlet_open_delay : TIMER;
   p21r10_timer_platen_open_delay : TIMER;
   p21r10_timer_press_cure : TIMER := (PRE := 55000);
   p21r10_timer_warning : TIMER[4];
   p21r11_index_kd : REAL;
   p21r11_index_ki : REAL := 0.1;
   p21r11_index_kp : REAL := 2.0;
   p21r11_run_kd : REAL;
   p21r11_run_ki : REAL := 0.8;
   p21r11_run_kp : REAL := 0.75;
   p21r16 : routine := (comment := -1073741697, oneshot := 1024);
   p21r16_pb_heater_off : BOOL;
   p21r16_pb_heater_on : BOOL;
   p21r16_permissive_run : BOOL := 1;
   p21r16_pid_temp_cv : REAL;
   p21r16_pid_temp_pv : REAL := 371.30002;
   p21r16_pid_timer : TIMER := (ACC := 30, EN := 1, DN := 1);
   p21r16_request_heat : BOOL;
   p21r16_timer_fault : TIMER[16] := ([2].PRE := 2000);
   p21r16_timer_warning : TIMER[16];
   p22_ai_amps : REAL;
   p22_ai_hz : REAL;
   p22_ai_speed : REAL;
   p22_ai_torque : REAL;
   p22_ai_ts1_lc : REAL := 13.332257;
   p22_ao_selected_speed : REAL;
   p22_ao_torque : REAL := 300.0;
   p22_ao_vfd : REAL;
   p22_control_word : INT := 2#0000_0100_0000_0110;
   p22_di_brake : BOOL := 1;
   p22_di_close_nip_roll : BOOL;
   p22_di_jog : BOOL;
   p22_di_jog_fwd : BOOL;
   p22_di_jog_rev : BOOL;
   p22_di_open_nip_roll : BOOL := 1;
   p22_di_run : BOOL := 1;
   p22_di_therm : BOOL := 1;
   p22_dint_to_hmi : DINT[16] := ([0] := 4, [1] := 4920, [2] := 5, [7] := 2);
   p22_do_close_nip_roll : BOOL;
   p22_param_ts1_jog_speed : REAL := 13.0;
   p22_real_to_hmi : REAL[112] := ([0] := 13.332517, [40] := 5.0, [41] := 2.0);
   p22_status_word : INT := 2#0001_0011_0011_1000;
   p22_ts1_acc_rate : REAL := 8.0;
   p22_ts1_decel_rate : REAL := 8.0;
   p22_ts1_gear_ratio : REAL := 54.76;
   p22_ts1_roll_diameter_ft : REAL := 0.5;
   p22_ts1_vfd : ABB_PROTOCOL_VFD := (STATUS_WORD := 4920, CONTROL_WORD := 1030, DRIVE_NOT_READY_FAULT := 1, OUT_FAULT := 1);
   p22_vfd_input_max : REAL := 2000.0;
   p22_vfd_input_min : REAL := -2000.0;
   p22_vfd_output_max : REAL := 20000.0;
   p22_vfd_output_min : REAL := -20000.0;
   p22r01 : routine := (comment := 7);
   p22r02 : routine := (comment := -1073741761);
   p22r02_fault_exists : BOOL := 1;
   p22r02_nip_open : BOOL := 1;
   p22r02_nip_open_dwell : TIMER := (PRE := 2000, ACC := 2020, EN := 1, DN := 1);
   p22r02_request_system_run : BOOL;
   p22r02_tension_dev_max : REAL := 75.0;
   p22r02_tension_dev_min : REAL := 45.0;
   p22r02_timer_fault : TIMER[4];
   p22r02_timer_warning : TIMER[4];
   p22r02_unack_fault : BOOL := 1;
   p22r02_unack_warning : BOOL;
   p22r02_warning_exists : BOOL;
   p22r03 : routine := (comment := -1073741761);
   p22r03_ave_tq : REAL;
   p22r03_hz : SYS_SCP := (Input_Max := 2000.0, Output_Max := 60.0);
   p22r03_lc_input_max : REAL := 10000.0;
   p22r03_lc_input_min : REAL;
   p22r03_lc_output_max : REAL := 250.0;
   p22r03_lc_output_min : REAL;
   p22r03_lc_scp : SYS_SCP := (Input := 533.68286, Input_Max := 10000.0, Output_Max := 250.0, Output := 13.342072);
   p22r03_sample_timer : TIMER := (PRE := 200, ACC := 123, EN := 1, TT := 1);
   p22r03_scaled_vfd_in : REAL;
   p22r03_timer_fault : TIMER[4];
   p22r03_timer_warning : TIMER[4];
   p22r03_tq_ave_ctrl : CONTROL := (LEN := 19);
   p22r03_tq_buffer : REAL[20];
   p22r03_tq_fifo : CONTROL := (LEN := 20, POS := 20, DN := 1);
   p22R03_ts1_vfd_rpm_to_speed : SYS_RPM_TO_SPEED := (IN_gear_ratio := 54.76, IN_roll_diameter := 0.5);
   p22r03_unload : DINT;
   p22r03_vfd_in_scaling : SYS_SCP := (Input_Min := -20000.0, Input_Max := 20000.0, Output_Min := -2000.0, Output_Max := 2000.0);
   p22r03_vfd_input_max : REAL := 20000.0;
   p22r03_vfd_input_min : REAL := -20000.0;
   p22r03_vfd_out_scaling : SYS_SCP := (Input_Min := -2000.0, Input_Max := 2000.0, Output_Min := -20000.0, Output_Max := 20000.0);
   p22r03_vfd_output_max : REAL := 2000.0;
   p22r03_vfd_output_min : REAL := -2000.0;
   p22r04 : routine := (comment := -1073741761);
   p22r04_speed_to_vfd_1 : SYS_SPEED_TO_VFD := (IN_gear_ratio := 54.76, IN_roll_diameter := 0.5);
   p22r04_timer_fault : TIMER[4];
   p22r04_timer_warning : TIMER[4];
   p22r05 : routine := (comment := -1073741761);
   p22r05_timer_fault : TIMER[4];
   p22r05_timer_warning : TIMER[4];
   p22r06 : routine := (comment := -1073741572);
   p22r06_ave_lc : REAL := 13.297389;
   p22r06_lc_buffer : REAL[20] := ([0] := 13.273371, [1] := 13.312629, [2] := 13.307721, [3] := 13.346979, [4] := 13.342072, [5] := 13.268463, [6] := 13.268463, [7] := 13.307721, [8] := 13.278277, [9] := 13.356793, [10] := 13.302814, [11] := 13.307721, [12] := 13.307721, [13] := 13.342072, [14] := 13.288093, [15] := 13.322443, [16] := 13.292999, [17] := 13.2635565, [18] := 13.292999, [19] := 13.361701);
   p22r06_lc_ctrl : CONTROL := (LEN := 20, POS := 20, DN := 1);
   p22r06_sample_timer : TIMER := (ACC := 31, EN := 1, DN := 1);
   p22r06_timer_fault : TIMER[4];
   p22r06_timer_warning : TIMER[4];
   p22r06_unload : DINT := 13;
   p22r07 : routine := (comment := -1073741761);
   p22r07_timer_fault : TIMER[4];
   p22r07_timer_warning : TIMER[4];
   p22r08 : routine := (comment := -1073741761);
   p22r08_timer_fault : TIMER[4];
   p22r08_timer_warning : TIMER[4];
   p22r09 : routine := (comment := -1073741761, fault := 1, fault_ack := 1);
   p22r09_mode_jog : BOOL;
   p22r09_mode_run : BOOL := 1;
   p22r09_mode_thread : BOOL;
   p22r09_pb_jog_fwd : BOOL;
   p22r09_pb_jog_rev : BOOL;
   p22r09_timer_fault : TIMER[4];
   p22r09_timer_warning : TIMER[4];
   p22r10 : routine := (comment := -1073741761);
   p22r10_calc_speed_offset : REAL;
   p22r10_param_psn_gain : REAL := 15.0;
   p22r10_pid_out : REAL := 50.0;
   p22r10_pid_psn : PID := (CTL := -1004502400, EN := 1, CT := 1, SWM := 1, NOBC := 1, INI := 1, DVPA := 1, PVHA := 1, SP := 60.0, KP := 5.0, KI := 2.0, BIAS := 1.0, MAXS := 500.0, SO := 50.0, MAXO := 100.0, UPD := 0.01, PV := 13.253741, ERR := 46.746258, OUT := 50.0, MAXI := 500.0, MAXCV := 100.0, MAXTIE := 100.0, DATA[0] := 2.2537422, DATA[1] := -42.411972, DATA[2] := 13.253741, DATA[3] := 46.746258, DATA[4] := 60.0, DATA[5] := 0.2, DATA[6] := 1.0, DATA[7] := 0.16, DATA[8] := 5.0, DATA[9] := 2.0, DATA[11] := 5.0, DATA[12] := 2.0, DATA[15] := 1.0, DATA[16] := 1.0);
   p22r10_pid_psn_cv : REAL := 50.0;
   p22r10_pid_psn_pv : REAL := 13.312629;
   p22r10_selected_torque : REAL := 300.0;
   p22r10_speed_offset : REAL;
   p22r10_stretch : REAL;
   p22r10_timer_fault : TIMER[4];
   p22r10_timer_warning : TIMER[4];
   p22r11 : routine := (comment := -1073741713, fault := 5, unack_fault := 1);
   p22r11_acc_decel_ramp : SYS_ACC_DEC_RAMP := (IN_param_master_accel_rate := 8.0, IN_param_master_decel_rate := 8.0, IN_last_scan_s := 0.03104);
   p22r11_permissive_jog : BOOL;
   p22r11_request_jog_fwd : BOOL;
   p22r11_request_jog_rev : BOOL;
   p22r11_request_line_jog : BOOL;
   p22r11_request_line_run : BOOL;
   p22r11_request_start : BOOL;
   p22r11_request_tension : BOOL;
   p22r11_request_thread_fwd : BOOL;
   p22r11_request_thread_rev : BOOL;
   p22r11_selected_speed : REAL;
   p22r11_timer_fault : TIMER[10] := ([0].PRE := 500, [0].ACC := 521, [0].EN := 1, [0].DN := 1, [2].PRE := 2000, [2].ACC := 2021, [2].EN := 1, [2].DN := 1);
   p22r11_timer_warning : TIMER[5] := ([1].PRE := 10000, [2].PRE := 10000);
   p22r11_zero_speed : BOOL := 1;
   p23_ai_lfl : REAL;
   p23_ai_metering_roll_amps : REAL;
   p23_ai_metering_roll_hz : REAL := 3.8146973e-06;
   p23_ai_metering_roll_speed_fpm : REAL;
   p23_ai_prs : REAL := -0.004393652;
   p23_ai_servo_ds_position : REAL := 0.008;
   p23_ai_servo_ds_torque : REAL := 6553.5;
   p23_ai_servo_ds_velocity : REAL;
   p23_ai_servo_os_position : REAL := 0.008;
   p23_ai_servo_os_torque : REAL := 7.0;
   p23_ai_servo_os_velocity : REAL;
   p23_ai_supply_amps : REAL;
   p23_ai_supply_hz : REAL := 60.0;
   p23_ai_supply_rpm : REAL;
   p23_ao_selected_speed : REAL;
   p23_ao_servo_ds_jog_vel_cmd : REAL := 0.003;
   p23_ao_servo_ds_position_cmd : REAL := 0.035;
   p23_ao_servo_ds_velocity_cmd : REAL := 0.0145;
   p23_ao_servo_ds_zero_offset : REAL := 0.036;
   p23_ao_servo_os_jog_vel_cmd : REAL := 0.003;
   p23_ao_servo_os_position_cmd : REAL := 0.035;
   p23_ao_servo_os_velocity_cmd : REAL := 0.0145;
   p23_ao_servo_os_zero_offset : REAL := 0.036;
   p23_ao_supply_selected_speed : REAL;
   p23_ave : CONTROL := (LEN := 9);
   p23_cpr_gear_ratio : REAL := 91.4;
   p23_cpr_roll_diameter_ft : REAL := 0.833;
   p23_cpr_speed_to_vfd : SYS_SPEED_TO_VFD := (IN_gear_ratio := 91.4, IN_roll_diameter := 0.833);
   p23_ctr_gear_ratio : REAL := 91.40625;
   p23_ctr_lfl_input_max : REAL := 30840.0;
   p23_ctr_lfl_input_min : REAL;
   p23_ctr_lfl_output_max : REAL := 100.0;
   p23_ctr_lfl_output_min : REAL;
   p23_ctr_roll_diameter_ft : REAL := 0.8333;
   p23_di_exhaust_speed_ok : BOOL;
   p23_di_filter_clean : BOOL := 1;
   p23_di_impreg_exhaust_running : BOOL;
   p23_di_impreg_tank_up : BOOL;
   p23_di_metering_bar_close : BOOL;
   p23_di_metering_bar_open : BOOL;
   p23_di_metering_roll : acs800_di_normal := (ready := 1, ctrl_from_net := 1, ref_from_net := 1, at_reference := 1);
   p23_di_servo_ds : servo_di := (mode_bit_1 := 1, homed := 1, stand_still := 1, drive_does_not_follow := 1, class_3_diagnostic := 1, operation_bit_15 := 1);
   p23_di_servo_os : servo_di := (mode_bit_1 := 1, homed := 1, stand_still := 1, drive_does_not_follow := 1, class_3_diagnostic := 1, operation_bit_15 := 1);
   p23_di_splice_jump : BOOL;
   p23_di_spring : acs800_di_normal := (ready := 1, ctrl_from_net := 1, ref_from_net := 1, at_reference := 1);
   p23_di_srv_ds_ok : BOOL;
   p23_di_srv_op_ok : BOOL := 1;
   p23_di_supply : acs800_di_normal := (ready := 1, ctrl_from_net := 1, ref_from_net := 1);
   p23_di_supply_motor_therm : BOOL := 1;
   p23_di_supply_speed_ok : BOOL;
   p23_di_tank_level_high : BOOL;
   p23_di_tank_level_low : BOOL;
   p23_di_therm : BOOL := 1;
   p23_di_though_level_low : BOOL;
   p23_di_vfd_jog_fwd : BOOL;
   p23_di_vfd_jog_rev : BOOL;
   p23_dint_to_hmi : DINT[32] := ([1] := 33845488, [3] := 207668736, [4] := 4352, [5] := 2, [6] := 2, [7] := 3, [10] := -1, [11] := -1, [12] := -1, [13] := -1);
   p23_do_enable_impreg_exhaust_fan : BOOL;
   p23_do_enable_impreg_supply_fan : BOOL;
   p23_do_impreg : acs800_do_normal;
   p23_do_impreg_nip_close : BOOL;
   p23_do_servo_ds : servo_do;
   p23_do_servo_os : servo_do;
   p23_do_Spring : acs800_do_normal;
   p23_do_supply : acs800_do_normal;
   p23_mtr_acc_rate : REAL := 15.0;
   p23_mtr_decel_rate : REAL := 15.0;
   p23_param_lfl_hhl : REAL := 30.0;
   p23_param_lfl_hl : REAL := 10.0;
   p23_param_min_start_tension : REAL := 20.0;
   p23_param_minus_adj_rate : REAL := -0.4;
   p23_param_mtr_jog_speed : REAL := 13.0;
   p23_param_plus_adj_rate : REAL := 1.0;
   p23_param_zone_pressure : REAL := -0.25;
   p23_real_to_hmi : REAL[112] := ([0] := 0.014, [1] := 0.014, [2] := 0.003, [3] := 0.0145, [8] := 3.8146973e-06, [11] := 60.0, [17] := 6553.4, [22] := 0.008, [23] := 2.0, [28] := -0.004069388, [55] := 10.0, [56] := 30.0, [58] := -0.25, [60] := 0.008, [61] := 0.008);
   p23_servo_ds_error : SYS_ENC_WITH_ZERO_BIT := (OUT_Status := -1);
   p23_servo_ds_warning : SYS_ENC_WITH_ZERO_BIT := (OUT_Status := -1);
   p23_servo_os_error : SYS_ENC_WITH_ZERO_BIT := (OUT_Status := -1);
   p23_servo_os_warning : SYS_ENC_WITH_ZERO_BIT := (OUT_Status := -1);
   p23_spring_gear_ratio : REAL := 145.0;
   p23_spring_roll_diameter_ft : REAL := 0.5;
   p23_spring_speed_to_vfd : SYS_SPEED_TO_VFD := (IN_gear_ratio := 145.0, IN_roll_diameter := 0.5);
   p23r01 : routine := (comment := 7);
   p23r02 : routine := (comment := -1073741761);
   p23r02_fault_exists : BOOL;
   p23r02_pb_start_exh : BOOL;
   p23r02_pb_stop_exh : BOOL;
   p23r02_request_nip_close : BOOL;
   p23r02_timer_fault : TIMER[4] := ([1].PRE := 2000);
   p23r02_timer_warning : TIMER[4] := ([1].PRE := 1000, [3].PRE := 5000);
   p23r02_unack_fault : BOOL;
   p23r02_unack_warning : BOOL := 1;
   p23r02_warning_exists : BOOL := 1;
   p23r03 : routine := (comment := -1073741793);
   p23r03_hz : SYS_SCP := (Input_Max := 1750.0, Output_Max := 60.0, Output := 3.8146973e-06);
   p23r03_impreg_lfl_monitor : SYS_SCP := (Input_Max := 30840.0, Output_Max := 100.0);
   p23r03_impreg_prs_input_max : REAL := 30840.0;
   p23r03_impreg_prs_input_min : REAL;
   p23r03_impreg_prs_output_max : REAL := 0.25;
   p23r03_impreg_prs_output_min : REAL := -0.25;
   p23r03_impreg_prs_scp : SYS_SCP := (Input := 15189.0, Input_Max := 30840.0, Output_Min := -0.25, Output_Max := 0.25, Output := -0.0037451386);
   p23r03_metering_vfd_rpm_to_speed : SYS_RPM_TO_SPEED := (IN_gear_ratio := 91.40625, IN_roll_diameter := 0.8333);
   p23r03_timer_fault : TIMER[4];
   p23r03_timer_warning : TIMER[4];
   p23r04 : routine := (comment := -1073741793);
   p23r04_timer_fault : TIMER[4];
   p23r04_timer_warning : TIMER[4];
   p23r05 : routine := (comment := -1073741761);
   p23r05_supply_status : DINT := 3;
   p23r05_timer_fault : TIMER[4];
   p23r05_timer_warning : TIMER[4];
   p23r06 : routine := (comment := -1073741796);
   p23r06_timer_fault : TIMER[4];
   p23r06_timer_warning : TIMER[4];
   p23r07 : routine := (comment := -1073741761);
   p23r07_timer_fault : TIMER[4];
   p23r07_timer_warning : TIMER[4];
   p23r08 : routine := (comment := -1073741761);
   p23r08_timer_fault : TIMER[4];
   p23r08_timer_warning : TIMER[4];
   p23r09 : routine := (comment := -1073741761);
   p23r09_mode_run : BOOL := 1;
   p23r09_timer_fault : TIMER[4];
   p23r09_web_wet_ctrl_toggle : SYS_Toggle := (toggle_state := 1);
   p23r10 : routine := (comment := -1073741761);
   p23r10_timer_fault : TIMER[4];
   p23r10_timer_warning : TIMER[4];
   p23r11 : routine := (comment := -1073741698, warning := 1, unack_warning := 1);
   p23r11_impreg_gap_os : REAL := 0.0175;
   p23r11_offsets : REAL[100] := ([8] := 0.0002, [12] := 0.0002, [13] := 0.0002, [14] := 0.0002, [15] := 0.0002, [16] := 0.0002, [17] := 0.0002, [18] := 0.0002);
   p23r11_permissive_jog : BOOL := 1;
   p23r11_pos_offset : REAL;
   p23r11_request_jog_fwd : BOOL;
   p23r11_request_jog_rev : BOOL;
   p23r11_request_position : BOOL;
   p23r11_request_start : BOOL;
   p23r11_request_zero : BOOL;
   p23r11_selected_position : REAL := 0.0175;
   p23r11_servo_not_ready : BOOL;
   p23r11_servo_status_ab : BOOL := 1;
   p23r11_servo_status_af : BOOL;
   p23r11_servo_status_bb : BOOL;
   p23r11_timer : TIMER[4] := ([0].ACC := 31, [0].EN := 1, [0].DN := 1);
   p23r11_timer_fault : TIMER[4];
   p23r11_timer_warning : TIMER[4];
   p23r12 : routine := (comment := -1073741698, warning := 1, unack_warning := 1);
   p23r12_impreg_gap_ds : REAL := 0.0175;
   p23r12_offsets : REAL[100] := ([8] := 0.0002, [12] := 0.0002, [13] := 0.0002, [14] := 0.0002, [15] := 1.e-04, [16] := 1.e-04, [17] := 1.e-04, [18] := 1.e-04);
   p23r12_permissive_jog : BOOL := 1;
   p23r12_pos_offset : REAL;
   p23r12_request_jog_fwd : BOOL;
   p23r12_request_jog_rev : BOOL;
   p23r12_request_position : BOOL;
   p23r12_request_start : BOOL;
   p23r12_request_zero : BOOL;
   p23r12_selected_position : REAL := 0.0175;
   p23r12_servo_not_ready : BOOL;
   p23r12_servo_status_ab : BOOL := 1;
   p23r12_servo_status_af : BOOL;
   p23r12_servo_status_bb : BOOL;
   p23r12_timer : TIMER[4] := ([0].ACC := 30, [0].EN := 1, [0].DN := 1);
   p23r12_timer_fault : TIMER[4];
   p23r12_timer_warning : TIMER[4];
   p23r13 : routine := (comment := -1073741697, oneshot := 1);
   p23r13_pb_start : BOOL;
   p23r13_pb_stop : BOOL;
   p23r13_request_auto_run : BOOL;
   p23r13_run_permissive : BOOL := 1;
   p23r13_timer_fault : TIMER[10] := ([5].PRE := 5000);
   p23r13_timer_warning : TIMER[4] := ([1].PRE := 1000, [2].PRE := 10000);
   p23r13_vfd_stopped : BOOL := 1;
   p23r15 : routine := (comment := -1073741713);
   p23r15_acc_decel_ramp : SYS_ACC_DEC_RAMP := (IN_param_master_accel_rate := 15.0, IN_param_master_decel_rate := 15.0, IN_last_scan_s := 0.030604);
   p23r15_adjust_dwell1 : TIMER := (PRE := 20000);
   p23r15_average_tension : REAL := 58.436848;
   p23r15_dead_band_minus : REAL := 55.0;
   p23r15_dead_band_plus : REAL := 65.0;
   p23r15_dead_band_setpoint : REAL := 5.0;
   p23r15_debounce_timer : TIMER := (PRE := 2000, ACC := 2000);
   p23r15_ffl : CONTROL := (LEN := 10, POS := 9);
   p23r15_ffu_temp : REAL := 56.845432;
   p23r15_fll_stack : REAL[50] := ([0] := 55.962414, [1] := 58.927414, [2] := 57.3234, [3] := 59.008427, [4] := 60.847378, [5] := 57.64744, [6] := 58.044395, [7] := 57.963383, [8] := 60.20739, [10] := 108.79131, [11] := 101.68503, [12] := 100.24141, [13] := 100.53305, [14] := 105.432594, [15] := 103.07518, [16] := 106.29294, [17] := 103.507774, [18] := 102.11763, [20] := 103.94038, [21] := 99.57064, [22] := 100.149055, [23] := 101.106606, [24] := 99.040825, [25] := 99.71646, [26] := 98.370056, [27] := 101.34964, [28] := 96.83409, [29] := 100.43584, [30] := 96.83409, [31] := 98.60823, [32] := 99.90603, [33] := 99.76507, [34] := 101.53921, [35] := 98.60823, [36] := 102.02042, [37] := 100.917046, [38] := 106.676926);
   p23r15_mean_adjust_acitve : BOOL;
   p23r15_minus_adjust : REAL := 1.0;
   p23r15_minus_adjust_acitve : BOOL;
   p23r15_minus_offset : REAL := -0.4;
   p23r15_neutral_offset : REAL := 0.4;
   p23r15_permissive_jog : BOOL := 1;
   p23r15_permissive_run : BOOL;
   p23r15_pid_tension_control : BOOL := 1;
   p23r15_plus_adjust : REAL := 1.0;
   p23r15_plus_adjust_acitve : BOOL;
   p23r15_plus_offset : REAL := 1.0;
   p23r15_request_jog_fwd : BOOL;
   p23r15_request_jog_rev : BOOL;
   p23r15_request_line_run : BOOL;
   p23r15_request_thread_fwd : BOOL;
   p23r15_request_thread_rev : BOOL;
   p23r15_sample_timer : TIMER := (PRE := 100);
   p23r15_selected_speed : REAL;
   p23r15_timer_fault : TIMER[10];
   p23r15_timer_warning : TIMER[5] := ([0].PRE := 30000);
   p23r15_ts1_tension_ok : BOOL;
   p23r15_zero_speed : BOOL := 1;
   p23r17_acc_decel_ramp : SYS_ACC_DEC_RAMP;
   p23r17_adjusted_speed : REAL;
   p23r17_ao_selected_speed : REAL;
   p23r17_di_brake : BOOL := 1;
   p23r17_di_therm : BOOL := 1;
   p23r17_hmi_vfd_jog_fwd : BOOL := 1;
   p23r17_permissive_jog : BOOL := 1;
   p23r17_permissive_run : BOOL;
   p23r17_request_jog_fwd : BOOL;
   p23r17_request_jog_rev : BOOL;
   p23r17_request_thread_fwd : BOOL;
   p23r17_request_thread_rev : BOOL;
   p23r17_sample_timer : TIMER := (PRE := 100);
   p23r17_selected_speed : REAL;
   p23r17_spd_adj : REAL;
   p23r17_sprng_assist_hmi_auto : BOOL := 1;
   p23r17_sprng_assist_hmi_jog : BOOL;
   p23r17_timer_fault : TIMER[10] := ([2].PRE := 3000);
   p23r17_timer_warning : TIMER[5];
   p23r17_zero_speed : BOOL := 1;
   p24_di_edge_guide_auto : BOOL := 1;
   p24_di_edge_guide_center : BOOL := 1;
   p24_di_edge_guide_left : BOOL := 1;
   p24_di_edge_guide_right : BOOL;
   p24_dint_to_hmi : DINT[16];
   p24_do_edge_guide_input_1 : BOOL := 1;
   p24_do_edge_guide_input_2 : BOOL;
   p24_do_edge_guide_input_3 : BOOL;
   p24_do_edge_guide_input_4 : BOOL;
   p24_do_edge_guide_input_5 : BOOL;
   p24_real_to_hmi : REAL[112];
   p24r01 : routine := (comment := 7);
   p24r02 : routine := (comment := -1073741761);
   p24r02_fault_exists : BOOL;
   p24r02_timer_fault : TIMER[4];
   p24r02_timer_warning : TIMER[4];
   p24r02_unack_fault : BOOL;
   p24r02_unack_warning : BOOL;
   p24r02_warning_exists : BOOL;
   p24r03 : routine := (comment := -1073741761);
   p24r03_timer_fault : TIMER[4];
   p24r03_timer_warning : TIMER[4];
   p24r04 : routine := (comment := -1073741809);
   p24r04_timer_fault : TIMER[4];
   p24r04_timer_warning : TIMER[4];
   p24r05 : routine := (comment := -1073741809);
   p24r05_timer_fault : TIMER[4];
   p24r05_timer_warning : TIMER[4];
   p24r06 : routine := (comment := -1073741793);
   p24r06_timer_fault : TIMER[4];
   p24r06_timer_warning : TIMER[4];
   p24r07 : routine := (comment := -1073741761);
   p24r07_timer_fault : TIMER[4];
   p24r07_timer_warning : TIMER[4];
   p24r08 : routine := (comment := -1073741761);
   p24r08_timer_fault : TIMER[4];
   p24r08_timer_warning : TIMER[4];
   p24r09 : routine := (comment := -1073741761);
   p24r09_timer_fault : TIMER[4];
   p24r09_timer_warning : TIMER[4];
   p24r10 : routine := (comment := -1073741761);
   p24r10_edge_guide_auto_request : BOOL := 1;
   p24r10_edge_guide_center_request : BOOL;
   p24r10_edge_guide_jog_left_request : BOOL;
   p24r10_edge_guide_jog_right_request : BOOL;
   p24r10_timer_fault : TIMER[4];
   p24r10_timer_warning : TIMER[4];
   p25_ai_amps : DINT;
   p25_ai_hz : DINT;
   p25_ai_rpm : REAL;
   p25_ai_speed : REAL;
   p25_ai_torque : REAL;
   p25_ai_ts2_lc : REAL;
   p25_ao_selected_speed : REAL;
   p25_ao_torque : REAL := 300.0;
   p25_ao_vfd : REAL;
   p25_control_word : INT := 2#0000_0100_0000_0110;
   p25_di_brake : BOOL := 1;
   p25_di_jog : BOOL;
   p25_di_jog_fwd : BOOL;
   p25_di_jog_rev : BOOL;
   p25_di_run : BOOL := 1;
   p25_di_therm : BOOL := 1;
   p25_di_ts2 : acs800_di_normal := (ready := 1, ctrl_from_net := 1, ref_from_net := 1, at_reference := 1);
   p25_dint_to_hmi : DINT[16] := ([0] := 983808, [1] := 4920, [2] := 5, [6] := 131072, [7] := 2);
   p25_param_ts2_jog_speed : REAL := 13.0;
   p25_real_to_hmi : REAL[112] := ([40] := 3.2, [41] := 0.5);
   p25_status_word : INT := 2#0001_0011_0011_1000;
   p25_ts2_acc_rate : REAL := 8.0;
   p25_ts2_decel_rate : REAL := 8.0;
   p25_ts2_gear_ratio : REAL := 108.75;
   p25_ts2_roll_diameter_ft : REAL := 1.0;
   p25_ts2_vfd : ABB_PROTOCOL_VFD := (STATUS_WORD := 4920, CONTROL_WORD := 1030, DRIVE_NOT_READY_FAULT := 1, OUT_FAULT := 1);
   p25_vfd_input_max : REAL := 2000.0;
   p25_vfd_input_min : REAL := -2000.0;
   p25_vfd_output_max : REAL := 20000.0;
   p25_vfd_output_min : REAL := -20000.0;
   p25r01 : routine := (comment := 7);
   p25r02 : routine := (comment := -1073741761);
   p25r02_fault_exists : BOOL := 1;
   p25r02_tension_dev_max : REAL := 75.0;
   p25r02_tension_dev_min : REAL := 45.0;
   p25r02_timer_fault : TIMER[4];
   p25r02_timer_warning : TIMER[4];
   p25r02_unack_fault : BOOL := 1;
   p25r02_unack_warning : BOOL;
   p25r02_warning_exists : BOOL;
   p25r03 : routine := (comment := -1073741761);
   p25r03_ave_tq : REAL;
   p25r03_hz : SYS_SCP := (Input_Max := 2000.0, Output_Max := 60.0);
   p25r03_lc_input_max : REAL := 30860.0;
   p25r03_lc_input_min : REAL;
   p25r03_lc_output_max : REAL := 250.0;
   p25r03_lc_output_min : REAL;
   p25r03_lc_scp : SYS_SCP := (Input_Max := 30860.0, Output_Max := 250.0);
   p25r03_sample_timer : TIMER := (PRE := 200, EN := 1, TT := 1);
   p25r03_scaled_vfd_in : REAL;
   p25r03_timer_fault : TIMER[4];
   p25r03_timer_warning : TIMER[4];
   p25r03_tq_ave_ctrl : CONTROL := (LEN := 19);
   p25r03_tq_buffer : REAL[20];
   p25r03_tq_fifo : CONTROL := (LEN := 20, POS := 20, DN := 1);
   p25R03_ts2_vfd_rpm_to_speed : SYS_RPM_TO_SPEED := (IN_gear_ratio := 108.75, IN_roll_diameter := 1.0);
   p25r03_unload : DINT;
   p25r03_vfd_in_scaling : SYS_SCP := (Input_Min := -20000.0, Input_Max := 20000.0, Output_Min := -2000.0, Output_Max := 2000.0);
   p25r03_vfd_input_max : REAL := 20000.0;
   p25r03_vfd_input_min : REAL := -20000.0;
   p25r03_vfd_out_scaling : SYS_SCP := (Input_Min := -2000.0, Input_Max := 2000.0, Output_Min := -20000.0, Output_Max := 20000.0);
   p25r03_vfd_output_max : REAL := 2000.0;
   p25r03_vfd_output_min : REAL := -2000.0;
   p25r04 : routine := (comment := -1073741761);
   p25r04_speed_to_vfd_ts2_scp : SYS_SPEED_TO_VFD := (IN_gear_ratio := 108.75, IN_roll_diameter := 1.0);
   p25r04_timer_fault : TIMER[4];
   p25r04_timer_warning : TIMER[4];
   p25r05 : routine := (comment := -1073741761);
   p25r05_timer_fault : TIMER[4];
   p25r05_timer_warning : TIMER[4];
   p25r06 : routine := (comment := -1073741572);
   p25r06_ave_lc : REAL;
   p25r06_lc_ave_ctrl : CONTROL := (LEN := 19);
   p25r06_lc_buffer : REAL[20];
   p25r06_lc_ctrl : CONTROL := (LEN := 20, POS := 20, DN := 1);
   p25r06_sample_timer : TIMER := (PRE := 200, ACC := 91, EN := 1, TT := 1);
   p25r06_timer_fault : TIMER[4];
   p25r06_timer_warning : TIMER[4];
   p25r06_unload : REAL;
   p25r07 : routine := (comment := -1073741761);
   p25r07_timer_fault : TIMER[4];
   p25r07_timer_warning : TIMER[4];
   p25r08 : routine := (comment := -1073741761);
   p25r08_timer_fault : TIMER[4];
   p25r08_timer_warning : TIMER[4];
   p25r09 : routine := (comment := -1073741761);
   p25r09_mode_jog : BOOL;
   p25r09_mode_run : BOOL := 1;
   p25r09_mode_thread : BOOL;
   p25r09_pb_jog_fwd : BOOL;
   p25r09_pb_jog_rev : BOOL;
   p25r09_timer_fault : TIMER[4];
   p25r09_timer_warning : TIMER[4];
   p25r10 : routine := (comment := -1073741761);
   p25r10_calc_speed_offset : REAL;
   p25r10_param_psn_gain : REAL := 15.0;
   p25r10_pid_manual_request : BOOL := 1;
   p25r10_pid_out : REAL := 50.0;
   p25r10_pid_psn : PID := (CTL := -2078243968, EN := 1, SWM := 1, NOBC := 1, INI := 1, DVPA := 1, PVLA := 1, PVHA := 1, SP := 60.0, KP := 3.2, KI := 0.5, BIAS := 1.0, MAXS := 500.0, SO := 50.0, MAXO := 100.0, UPD := 0.01, ERR := 60.0, OUT := 50.0, MAXI := 500.0, MAXCV := 100.0, MAXTIE := 100.0, DATA[0] := 10.599998, DATA[3] := 60.0, DATA[4] := 60.0, DATA[5] := 0.2, DATA[6] := 1.0, DATA[7] := 0.16, DATA[8] := 3.2, DATA[9] := 0.5, DATA[11] := 3.2, DATA[12] := 0.5, DATA[15] := 1.0, DATA[16] := 1.0);
   p25r10_pid_psn_cv : REAL := 50.0;
   p25r10_pid_psn_pv : REAL;
   p25r10_speed_offset : REAL;
   p25r10_tension_request : BOOL;
   p25r10_timer_fault : TIMER[4];
   p25r10_timer_warning : TIMER[4];
   p25r11 : routine := (comment := -1073741713, fault := 5, unack_fault := 1);
   p25r11_acc_decel_ramp : SYS_ACC_DEC_RAMP := (IN_param_master_accel_rate := 8.0, IN_param_master_decel_rate := 8.0, IN_last_scan_s := 0.031384);
   p25r11_at_zero : BOOL := 1;
   p25r11_permissive_jog_thread : BOOL;
   p25r11_request_jog_fwd : BOOL;
   p25r11_request_jog_rev : BOOL;
   p25r11_request_line_jog : BOOL;
   p25r11_request_line_run : BOOL;
   p25r11_request_thread_fwd : BOOL;
   p25r11_request_thread_rev : BOOL;
   p25r11_selected_speed : REAL;
   p25r11_timer_fault : TIMER[10] := ([0].PRE := 500, [0].ACC := 521, [0].EN := 1, [0].DN := 1, [2].PRE := 2000, [2].ACC := 2021, [2].EN := 1, [2].DN := 1);
   p25r11_timer_warning : TIMER[4] := ([1].PRE := 10000, [2].PRE := 10000);
   p25r11_vfd_start_request : BOOL;
   p26_ao_dia_a : REAL := -75.37109;
   p26_ao_dia_b : REAL := -85.5;
   p26_dint_to_hmi : DINT[16] := ([0] := 5);
   p26_inactive_tension_sp : REAL;
   p26_ltf_a_sensor_input_max : REAL := 30959.0;
   p26_ltf_a_sensor_input_min : REAL := 100.0;
   p26_ltf_a_sensor_output_max : REAL := 55.0;
   p26_ltf_a_sensor_output_min : REAL := 4.0;
   p26_ltf_b_sensor_input_max : REAL := 30959.0;
   p26_ltf_b_sensor_input_min : REAL := 400.0;
   p26_ltf_b_sensor_output_max : REAL := 55.0;
   p26_ltf_b_sensor_output_min : REAL := 4.0;
   p26_real_to_hmi : REAL[112] := ([0] := -75.404144, [1] := -85.5);
   p26_ula_prs_input_max : REAL := 20.0;
   p26_ula_prs_input_min : REAL := 3.5;
   p26_ula_prs_output_max : REAL := 30840.0;
   p26_ula_prs_output_min : REAL := 5397.0;
   p26_ulb_prs_input_max : REAL := 20.0;
   p26_ulb_prs_input_min : REAL := 3.5;
   p26_ulb_prs_output_max : REAL := 30840.0;
   p26_ulb_prs_output_min : REAL := 5397.0;
   p26r01 : routine := (comment := 7);
   p26r02 : routine := (comment := -1073741761);
   p26r02_fault_exists : BOOL;
   p26r02_timer_fault : TIMER[4];
   p26r02_timer_warning : TIMER[4];
   p26r02_unack_fault : BOOL;
   p26r02_unack_warning : BOOL;
   p26r02_warning_exists : BOOL;
   p26r03 : routine := (comment := -1073741761);
   p26r03_a_radius : REAL := -37.685547;
   p26r03_ai_dia_a_sensor : REAL := 54.952072;
   p26r03_ai_dia_b_sensor : REAL := 55.0;
   p26r03_b_radius : REAL := -42.75;
   p26r03_ltf_a_sensor_scp : SYS_SCP := (Input := 30930.0, Input_Min := 100.0, Input_Max := 30959.0, Output_Min := 4.0, Output_Max := 55.0, Output := 54.952072);
   p26r03_ltf_b_sensor_scp : SYS_SCP := (Input := 30969.0, Input_Min := 400.0, Input_Max := 30959.0, Output_Min := 4.0, Output_Max := 55.0, Output := 55.0);
   p26r03_timer_fault : TIMER[4];
   p26r03_timer_warning : TIMER[4];
   p26r03_upper_A_tension_on : BOOL := 1;
   p26r03_upper_B_tension_on : BOOL := 1;
   p26r03_upper_poly_a_distance : REAL := 17.25;
   p26r03_upper_poly_b_distance : REAL := 12.25;
   p26r04 : routine := (comment := -1073741761);
   p26r04_timer_fault : TIMER[4];
   p26r04_timer_warning : TIMER[4];
   p26r04_ula_prs_scp : SYS_SCP := (Input := -75.37109, Input_Min := 3.5, Input_Max := 20.0, Output_Min := 5397.0, Output_Max := 30840.0, Output := 5397.0);
